KUKA KRL program: MyProgram_072().src

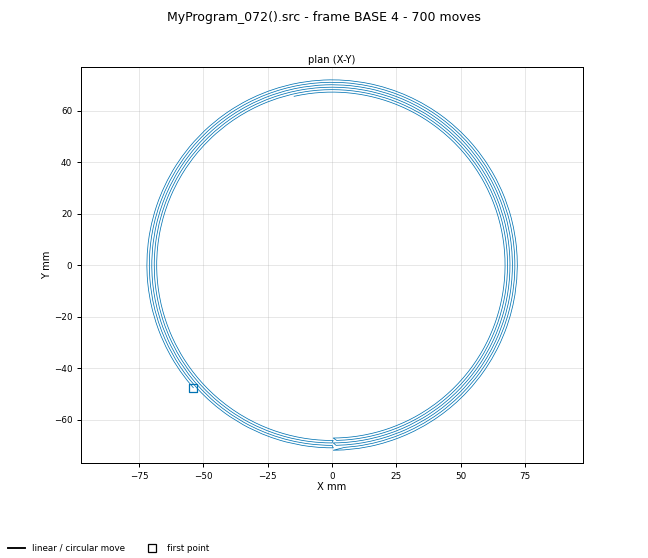
[picture p0: tool path of MyProgram_072().src in frame BASE 4, 700 of 700 moves have a stored position in this frame; points joined in program order, loops and branches not executed]
&ACCESS RVP
&REL 1
&PARAM TEMPLATE = C:\KRC\Roboter\Template\vorgabe
&PARAM EDITMASK = *
DEF MyProgram_072()
; ---- Setting reference (Base) ----
$BASE = BASE_DATA[4]

; --------------------------
; ---- Setting tool (TCP) ----
$TOOL = TOOL_DATA[3]
; --------------------------

$VEL.CP = VEL_APROX_PRINT
Startdeposition()
$VEL.CP = VEL_PRINT
LIN {X -53.9187,Y -47.6448,Z 77,A -144.3858,B 24.9058,C -2.2406,E1 24.8791,E2 228.8323} C_DIS
LIN {X -56.3583,Y -44.7314,Z 77,A -147.3901,B 24.9052,C -2.2481,E1 24.8738,E2 231.8326} C_DIS
LIN {X -58.9151,Y -41.3065,Z 77,A -151.2625,B 24.9054,C -2.2457,E1 24.8674,E2 235.7295} C_DIS
LIN {X -61.4241,Y -37.4729,Z 77,A -154.4026,B 24.9036,C -2.2665,E1 24.8627,E2 238.8358} C_DIS
LIN {X -62.7238,Y -35.2532,Z 77,A -157.5518,B 24.9052,C -2.2474,E1 24.8584,E2 242.0471} C_DIS
LIN {X -64.5699,Y -31.7477,Z 77,A -159.6161,B 24.9025,C -2.2803,E1 24.8558,E2 244.0442} C_DIS
LIN {X -66.4605,Y -27.5735,Z 77,A -163.4241,B 24.9019,C -2.2869,E1 24.8515,E2 247.8572} C_DIS
LIN {X -67.4022,Y -25.1814,Z 77,A -165.8052,B 24.902,C -2.2855,E1 24.8491,E2 250.2552} C_DIS
LIN {X -68.4094,Y -22.3006,Z 77,A -169.291,B 24.9034,C -2.2696,E1 24.8461,E2 253.7987} C_DIS
LIN {X -69.7872,Y -17.5225,Z 77,A -172.3901,B 24.9007,C -2.3002,E1 24.844,E2 256.8429} C_DIS
LIN {X -70.5609,Y -14.087,Z 77,A -174.6218,B 24.8989,C -2.3213,E1 24.8427,E2 259.0373} C_DIS
LIN {X -71.303,Y -9.6528,Z 77,A -178.4757,B 24.8985,C -2.3264,E1 24.841,E2 262.9021} C_DIS
LIN {X -71.6429,Y -6.6659,Z 77,A 179.1463,B 24.8978,C -2.3342,E1 24.8403,E2 265.2756} C_DIS
LIN {X -71.8296,Y -4.1964,Z 77,A 176.9907,B 24.8976,C -2.3365,E1 24.8399,E2 267.4388} C_DIS
LIN {X -71.951,Y -0.3995,Z 77,A 174.0055,B 24.8967,C -2.3469,E1 24.8398,E2 270.417} C_DIS
LIN {X -71.8201,Y 4.377,Z 77,A 169.8234,B 24.8963,C -2.3508,E1 24.8403,E2 274.615} C_DIS
LIN {X -71.4314,Y 8.6465,Z 77,A 166.8704,B 24.8945,C -2.3716,E1 24.8412,E2 277.5359} C_DIS
LIN {X -71.0021,Y 11.6566,Z 77,A 164.4409,B 24.8938,C -2.3791,E1 24.8422,E2 279.962} C_DIS
LIN {X -70.158,Y 15.9702,Z 77,A 161.2467,B 24.8922,C -2.3968,E1 24.8439,E2 283.1327} C_DIS
LIN {X -68.9886,Y 20.438,Z 77,A 157.304,B 24.8917,C -2.4024,E1 24.8468,E2 287.0849} C_DIS
LIN {X -68.1942,Y 22.9497,Z 77,A 155.1243,B 24.8913,C -2.4071,E1 24.8487,E2 289.266} C_DIS
LIN {X -67.3704,Y 25.267,Z 77,A 152.6721,B 24.8917,C -2.4023,E1 24.8511,E2 291.7435} C_DIS
LIN {X -65.9392,Y 28.7951,Z 77,A 148.9517,B 24.8922,C -2.3965,E1 24.8553,E2 295.4983} C_DIS
LIN {X -64.0236,Y 32.8348,Z 77,A 146.9975,B 24.8881,C -2.442,E1 24.8576,E2 297.3545} C_DIS
LIN {X -61.8148,Y 36.8256,Z 77,A 142.8596,B 24.8881,C -2.4411,E1 24.8633,E2 301.5161} C_DIS
LIN {X -60.5259,Y 38.9069,Z 77,A 140.6625,B 24.8881,C -2.4411,E1 24.8666,E2 303.7244} C_DIS
LIN {X -58.295,Y 42.1781,Z 77,A 137.1152,B 24.8881,C -2.4409,E1 24.8723,E2 307.2896} C_DIS
LIN {X -55.5018,Y 45.7902,Z 77,A 134.103,B 24.886,C -2.4642,E1 24.8775,E2 310.2602} C_DIS
LIN {X -53.6001,Y 48.0016,Z 77,A 131.2102,B 24.8867,C -2.4573,E1 24.8829,E2 313.1825} C_DIS
LIN {X -49.6348,Y 52.0931,Z 77,A 127.3776,B 24.8842,C -2.4839,E1 24.8903,E2 316.9677} C_DIS
LIN {X -47.6713,Y 53.8958,Z 77,A 124.8505,B 24.8846,C -2.4796,E1 24.8956,E2 319.5154} C_DIS
LIN {X -43.8735,Y 57.0285,Z 77,A 120.3096,B 24.8851,C -2.4739,E1 24.9056,E2 324.0866} C_DIS
LIN {X -41.0352,Y 59.1037,Z 77,A 118.2193,B 24.8831,C -2.4956,E1 24.9103,E2 326.1323} C_DIS
LIN {X -38.3583,Y 60.8757,Z 77,A 115.8538,B 24.8822,C -2.5048,E1 24.9158,E2 328.4836} C_DIS
LIN {X -34.6979,Y 63.0348,Z 77,A 112.3188,B 24.882,C -2.5073,E1 24.9244,E2 332.0233} C_DIS
LIN {X -32.2967,Y 64.2967,Z 77,A 110.0047,B 24.882,C -2.5072,E1 24.9301,E2 334.3439} C_DIS
LIN {X -29.0979,Y 65.8072,Z 77,A 106.6833,B 24.8827,C -2.4996,E1 24.9386,E2 337.6914} C_DIS
LIN {X -24.7486,Y 67.5622,Z 77,A 103.033,B 24.8821,C -2.5065,E1 24.9481,E2 341.3329} C_DIS
LIN {X -20.7016,Y 68.9104,Z 77,A 99.6928,B 24.8816,C -2.5117,E1 24.957,E2 344.6667} C_DIS
LIN {X -15.683,Y 70.2223,Z 77,A 95.9494,B 24.8803,C -2.5248,E1 24.9671,E2 348.384} C_DIS
LIN {X -12.4973,Y 70.8591,Z 77,A 93.0822,B 24.8808,C -2.5201,E1 24.975,E2 351.2656} C_DIS
LIN {X -7.8682,Y 71.5218,Z 77,A 89.6803,B 24.8798,C -2.5301,E1 24.9844,E2 354.6461} C_DIS
LIN {X -3.2799,Y 71.8778,Z 77,A 86.0502,B 24.8796,C -2.5325,E1 24.9945,E2 358.2719} C_DIS
LIN {X -0.9009,Y 71.9479,Z 77,A 83.3153,B 24.8815,C -2.5123,E1 25.0023,E2 361.0549} C_DIS
LIN {X 2.7139,Y 71.9018,Z 77,A 81.3961,B 24.8792,C -2.5363,E1 25.0075,E2 362.9166} C_DIS
LIN {X 6.8293,Y 71.6278,Z 77,A 77.9201,B 24.8797,C -2.5313,E1 25.0172,E2 366.4027} C_DIS
LIN {X 12.1948,Y 70.9121,Z 77,A 73.7586,B 24.8795,C -2.534,E1 25.0286,E2 370.5543} C_DIS
LIN {X 15.6992,Y 70.2197,Z 77,A 70.7865,B 24.8799,C -2.5294,E1 25.0368,E2 373.5334} C_DIS
LIN {X 19.6301,Y 69.2227,Z 77,A 67.0407,B 24.8813,C -2.5142,E1 25.0469,E2 377.3093} C_DIS
LIN {X 23.9385,Y 67.8535,Z 77,A 63.9687,B 24.8803,C -2.5248,E1 25.055,E2 380.3501} C_DIS
LIN {X 27.7756,Y 66.3753,Z 77,A 59.8788,B 24.8826,C -2.5004,E1 25.0657,E2 384.4886} C_DIS
LIN {X 31.1771,Y 64.8469,Z 77,A 57.9313,B 24.8805,C -2.5236,E1 25.0705,E2 386.3762} C_DIS
LIN {X 34.6789,Y 63.0444,Z 77,A 54.1919,B 24.8823,C -2.5036,E1 25.0798,E2 390.1524} C_DIS
LIN {X 38.4793,Y 60.8002,Z 77,A 51.0432,B 24.8819,C -2.5081,E1 25.0872,E2 393.2807} C_DIS
LIN {X 41.7065,Y 58.632,Z 77,A 48.2934,B 24.8815,C -2.5123,E1 25.0935,E2 396.011} C_DIS
LIN {X 43.7846,Y 57.097,Z 77,A 46.1388,B 24.8821,C -2.5061,E1 25.0984,E2 398.1726} C_DIS
LIN {X 46.6873,Y 54.7488,Z 77,A 42.9748,B 24.8831,C -2.4954,E1 25.1052,E2 401.3498} C_DIS
LIN {X 50.2229,Y 51.5263,Z 77,A 39.1466,B 24.8839,C -2.4872,E1 25.113,E2 405.1818} C_DIS
LIN {X 52.9217,Y 48.7488,Z 77,A 36.3509,B 24.8838,C -2.4884,E1 25.1184,E2 407.9624} C_DIS
LIN {X 54.7222,Y 46.7185,Z 77,A 34.2514,B 24.8841,C -2.4853,E1 25.1223,E2 410.06} C_DIS
LIN {X 56.9046,Y 44.0342,Z 77,A 31.1783,B 24.8855,C -2.47,E1 25.1277,E2 413.1549} C_DIS
LIN {X 59.7877,Y 40.0337,Z 77,A 27.4574,B 24.8859,C -2.466,E1 25.1336,E2 416.8672} C_DIS
LIN {X 62.2247,Y 36.1293,Z 77,A 23.0825,B 24.8886,C -2.4367,E1 25.14,E2 421.2888} C_DIS
LIN {X 63.774,Y 33.3177,Z 77,A 20.7832,B 24.8886,C -2.4369,E1 25.143,E2 423.5756} C_DIS
LIN {X 65.8578,Y 28.9817,Z 77,A 17.4795,B 24.8882,C -2.441,E1 25.1468,E2 426.8518} C_DIS
LIN {X 67.0447,Y 26.1186,Z 77,A 14.8515,B 24.8892,C -2.4294,E1 25.1496,E2 429.4926} C_DIS
LIN {X 68.871,Y 20.8324,Z 77,A 10.385,B 24.8905,C -2.4159,E1 25.1535,E2 433.9658} C_DIS
LIN {X 69.6052,Y 18.2306,Z 77,A 8.074,B 24.8915,C -2.405,E1 25.1552,E2 436.2893} C_DIS
LIN {X 70.4525,Y 14.6153,Z 77,A 5.2404,B 24.892,C -2.3994,E1 25.1569,E2 439.1195} C_DIS
LIN {X 71.252,Y 10.0146,Z 77,A 2.1561,B 24.8914,C -2.406,E1 25.1583,E2 442.1703} C_DIS
LIN {X 71.6054,Y 7.0466,Z 77,A -0.7092,B 24.8933,C -2.3847,E1 25.1592,E2 445.0689} C_DIS
LIN {X 71.868,Y 3.4604,Z 77,A -3.831,B 24.8948,C -2.3683,E1 25.1597,E2 448.2109} C_DIS
LIN {X 71.9513,Y -0.3429,Z 77,A -6.9056,B 24.8957,C -2.3574,E1 25.1597,E2 451.293} C_DIS
LIN {X 71.7394,Y -5.5341,Z 77,A -11.1078,B 24.897,C -2.3424,E1 25.159,E2 455.5057} C_DIS
LIN {X 71.0278,Y -11.5028,Z 77,A -16.3322,B 24.8995,C -2.3149,E1 25.1569,E2 460.7642} C_DIS
LIN {X 70.2523,Y -15.5498,Z 77,A -18.4428,B 24.8975,C -2.3377,E1 25.1558,E2 462.8086} C_DIS
LIN {X 69.2248,Y -19.6231,Z 77,A -21.5617,B 24.8978,C -2.3337,E1 25.1536,E2 465.919} C_DIS
LIN {X 67.943,Y -23.6835,Z 77,A -24.9418,B 24.8987,C -2.3235,E1 25.1508,E2 469.304} C_DIS
LIN {X 67.0842,Y -26.0181,Z 77,A -27.7452,B 24.9013,C -2.2941,E1 25.1479,E2 472.1614} C_DIS
LIN {X 65.4629,Y -29.864,Z 77,A -30.3132,B 24.9003,C -2.3055,E1 25.1451,E2 474.6883} C_DIS
LIN {X 64.2104,Y -32.4692,Z 77,A -33.0533,B 24.9019,C -2.2863,E1 25.1417,E2 477.4591} C_DIS
LIN {X 61.9999,Y -36.5125,Z 77,A -36.9921,B 24.9035,C -2.2682,E1 25.1362,E2 481.4202} C_DIS
LIN {X 59.5766,Y -40.3456,Z 77,A -40.253,B 24.9035,C -2.268,E1 25.1312,E2 484.6654} C_DIS
LIN {X 57.5966,Y -43.1251,Z 77,A -42.6994,B 24.9035,C -2.2683,E1 25.1272,E2 487.0993} C_DIS
LIN {X 54.3876,Y -47.1084,Z 77,A -46.7073,B 24.9042,C -2.2595,E1 25.1201,E2 491.1094} C_DIS
LIN {X 51.4117,Y -50.3396,Z 77,A -50.3462,B 24.9053,C -2.2469,E1 25.1132,E2 494.7622} C_DIS
LIN {X 48.408,Y -53.2321,Z 77,A -53.6707,B 24.906,C -2.2391,E1 25.1064,E2 498.0915} C_DIS
LIN {X 45.7832,Y -55.5077,Z 77,A -56.6724,B 24.907,C -2.2264,E1 25.0999,E2 501.1116} C_DIS
LIN {X 43.0423,Y -57.6588,Z 77,A -59.2217,B 24.907,C -2.2268,E1 25.0943,E2 503.6508} C_DIS
LIN {X 39.929,Y -59.8578,Z 77,A -62.2452,B 24.9075,C -2.221,E1 25.0873,E2 506.6776} C_DIS
LIN {X 35.9325,Y -62.3378,Z 77,A -66.2637,B 24.9087,C -2.2068,E1 25.0777,E2 510.7173} C_DIS
LIN {X 31.9087,Y -64.4901,Z 77,A -69.8151,B 24.909,C -2.203,E1 25.0689,E2 514.2679} C_DIS
LIN {X 28.8413,Y -65.919,Z 77,A -72.2737,B 24.9088,C -2.2052,E1 25.0626,E2 516.7151} C_DIS
LIN {X 26.0215,Y -67.0829,Z 77,A -74.4572,B 24.9085,C -2.2084,E1 25.057,E2 518.8861} C_DIS
LIN {X 23.2742,Y -68.0848,Z 77,A -77.7414,B 24.9108,C -2.1802,E1 25.0482,E2 522.2308} C_DIS
LIN {X 19.8136,Y -69.1708,Z 77,A -79.4127,B 24.9085,C -2.2091,E1 25.0439,E2 523.8305} C_DIS
LIN {X 16.8729,Y -69.9462,Z 77,A -82.0355,B 24.9091,C -2.2013,E1 25.0368,E2 526.4678} C_DIS
LIN {X 14.9547,Y -70.3821,Z 77,A -83.9899,B 24.9101,C -2.1896,E1 25.0314,E2 528.4473} C_DIS
LIN {X 10.5522,Y -71.1757,Z 77,A -87.9511,B 24.9111,C -2.1767,E1 25.0204,E2 532.4353} C_DIS
LIN {X 4.5761,Y -71.8072,Z 77,A -92.5167,B 24.9109,C -2.1799,E1 25.0077,E2 536.9906} C_DIS
LIN {X 0.4767,Y -71.9366,Z 77,A -94.7077,B 24.9086,C -2.2068,E1 25.0018,E2 539.1173} C_DIS
Enddeposition()
LIN {X 0.4767,Y -71.9366,Z 77,A -94.7077,B 24.9086,C -2.2068,E1 25.0018,E2 539.1173} C_DIS
Startdeposition()
$VEL.CP = VEL_PRINT
LIN {X 4.8028,Y -70.8374,Z 77,A -90.3844,B 24.9054,C -2.2459,E1 25.0141,E2 534.7027} C_DIS
LIN {X 9.797,Y -70.3212,Z 77,A -87.1467,B 24.907,C -2.227,E1 25.0229,E2 531.5122} C_DIS
LIN {X 11.8985,Y -69.9962,Z 77,A -84.5588,B 24.9049,C -2.2512,E1 25.0302,E2 528.8694} C_DIS
LIN {X 15.8769,Y -69.2021,Z 77,A -81.1578,B 24.9044,C -2.2576,E1 25.0395,E2 525.4579} C_DIS
LIN {X 19.7248,Y -68.2062,Z 77,A -78.0106,B 24.9042,C -2.2594,E1 25.048,E2 522.3116} C_DIS
LIN {X 24.4836,Y -66.6453,Z 77,A -74.1651,B 24.9042,C -2.2592,E1 25.0581,E2 518.4743} C_DIS
LIN {X 28.2316,Y -65.1461,Z 77,A -70.4132,B 24.9027,C -2.2774,E1 25.0678,E2 514.6881} C_DIS
LIN {X 31.7235,Y -63.5191,Z 77,A -68.2259,B 24.9044,C -2.2572,E1 25.0732,E2 512.5547} C_DIS
LIN {X 35.7437,Y -61.348,Z 77,A -64.1814,B 24.903,C -2.2734,E1 25.0831,E2 508.4836} C_DIS
LIN {X 39.7187,Y -58.8511,Z 77,A -61.0974,B 24.9041,C -2.2613,E1 25.0902,E2 505.4384} C_DIS
LIN {X 42.4392,Y -56.9209,Z 77,A -58.4529,B 24.9037,C -2.2654,E1 25.0962,E2 502.7933} C_DIS
LIN {X 44.0637,Y -55.6723,Z 77,A -55.8093,B 24.9011,C -2.2965,E1 25.1022,E2 500.086} C_DIS
LIN {X 47.6747,Y -52.6136,Z 77,A -52.5448,B 24.9016,C -2.2896,E1 25.109,E2 496.8507} C_DIS
LIN {X 50.1301,Y -50.2801,Z 77,A -49.8672,B 24.9012,C -2.2945,E1 25.1143,E2 494.1727} C_DIS
LIN {X 52.5803,Y -47.7124,Z 77,A -46.9276,B 24.9004,C -2.3037,E1 25.1199,E2 491.2242} C_DIS
LIN {X 55.7281,Y -43.9931,Z 77,A -43.3118,B 24.9004,C -2.305,E1 25.1263,E2 487.6221} C_DIS
LIN {X 57.3663,Y -41.8346,Z 77,A -40.9757,B 24.8994,C -2.3151,E1 25.1302,E2 485.2733} C_DIS
LIN {X 59.8557,Y -38.1883,Z 77,A -37.1704,B 24.898,C -2.3318,E1 25.1362,E2 481.4474} C_DIS
LIN {X 62.6104,Y -33.4832,Z 77,A -33.0702,B 24.8976,C -2.3359,E1 25.1418,E2 477.3589} C_DIS
LIN {X 64.9521,Y -28.6765,Z 77,A -28.9167,B 24.8969,C -2.344,E1 25.1468,E2 473.2084} C_DIS
LIN {X 66.7625,Y -24.1621,Z 77,A -24.9117,B 24.8957,C -2.3582,E1 25.1509,E2 469.1921} C_DIS
LIN {X 68.1104,Y -20.0502,Z 77,A -21.6688,B 24.8953,C -2.3619,E1 25.1536,E2 465.9591} C_DIS
LIN {X 68.9713,Y -16.8514,Z 77,A -18.6869,B 24.8938,C -2.3791,E1 25.1557,E2 462.9537} C_DIS
LIN {X 69.826,Y -12.8621,Z 77,A -15.6337,B 24.8935,C -2.3826,E1 25.1574,E2 459.91} C_DIS
LIN {X 70.2378,Y -10.3839,Z 77,A -12.2641,B 24.8894,C -2.4278,E1 25.1588,E2 456.4534} C_DIS
LIN {X 70.7674,Y -5.7434,Z 77,A -10.2321,B 24.8928,C -2.3897,E1 25.1593,E2 454.5236} C_DIS
LIN {X 70.9871,Y -1.3604,Z 77,A -6.2727,B 24.8907,C -2.4128,E1 25.1598,E2 450.5329} C_DIS
LIN {X 70.983,Y 1.5815,Z 77,A -3.6125,B 24.8893,C -2.4286,E1 25.1597,E2 447.8514} C_DIS
LIN {X 70.8141,Y 5.1488,Z 77,A -0.9641,B 24.8891,C -2.431,E1 25.1592,E2 445.2131} C_DIS
LIN {X 70.4749,Y 8.6274,Z 77,A 1.5523,B 24.8891,C -2.4311,E1 25.1585,E2 442.7112} C_DIS
LIN {X 70.1756,Y 10.789,Z 77,A 3.8082,B 24.8873,C -2.4507,E1 25.1575,E2 440.4222} C_DIS
LIN {X 69.5035,Y 14.5026,Z 77,A 6.5362,B 24.8873,C -2.451,E1 25.1561,E2 437.7094} C_DIS
LIN {X 68.834,Y 17.4059,Z 77,A 8.6114,B 24.8874,C -2.449,E1 25.1548,E2 435.6511} C_DIS
LIN {X 68.2901,Y 19.4287,Z 77,A 11.0027,B 24.8851,C -2.474,E1 25.1529,E2 433.2144} C_DIS
LIN {X 66.7102,Y 24.3056,Z 77,A 14.6305,B 24.8853,C -2.4716,E1 25.1497,E2 429.6126} C_DIS
LIN {X 64.9023,Y 28.7903,Z 77,A 18.5475,B 24.8843,C -2.4832,E1 25.1455,E2 425.69} C_DIS
LIN {X 63.9127,Y 30.9228,Z 77,A 20.6659,B 24.8832,C -2.4947,E1 25.1429,E2 423.5558} C_DIS
LIN {X 62.7651,Y 33.1899,Z 77,A 22.6008,B 24.883,C -2.497,E1 25.1405,E2 421.6256} C_DIS
LIN {X 59.7783,Y 38.3089,Z 77,A 27.1898,B 24.8823,C -2.504,E1 25.1339,E2 417.0434} C_DIS
LIN {X 57.097,Y 42.2025,Z 77,A 30.7011,B 24.8823,C -2.5051,E1 25.1283,E2 413.5469} C_DIS
LIN {X 54.6084,Y 45.3755,Z 77,A 33.7833,B 24.8819,C -2.508,E1 25.123,E2 410.4722} C_DIS
LIN {X 52.0939,Y 48.2426,Z 77,A 37.6886,B 24.8791,C -2.5376,E1 25.1156,E2 406.5143} C_DIS
LIN {X 49.5448,Y 50.8573,Z 77,A 41.0558,B 24.8774,C -2.5553,E1 25.1089,E2 403.1193} C_DIS
LIN {X 47.0744,Y 53.1521,Z 77,A 42.7817,B 24.8795,C -2.5335,E1 25.1054,E2 401.4521} C_DIS
LIN {X 43.9657,Y 55.7497,Z 77,A 45.6849,B 24.8799,C -2.5297,E1 25.0993,E2 398.5689} C_DIS
LIN {X 40.834,Y 58.0839,Z 77,A 49.1667,B 24.8785,C -2.544,E1 25.0914,E2 395.0659} C_DIS
LIN {X 38.929,Y 59.3765,Z 77,A 51.056,B 24.8781,C -2.5478,E1 25.087,E2 393.1738} C_DIS
LIN {X 36.7766,Y 60.7331,Z 77,A 53.5141,B 24.8768,C -2.5617,E1 25.0811,E2 390.6906} C_DIS
LIN {X 33.4485,Y 62.6267,Z 77,A 56.6188,B 24.8764,C -2.5663,E1 25.0735,E2 387.584} C_DIS
LIN {X 30.2857,Y 64.2177,Z 77,A 59.5792,B 24.8758,C -2.5724,E1 25.066,E2 384.6169} C_DIS
LIN {X 27.2313,Y 65.5714,Z 77,A 62.7226,B 24.8743,C -2.587,E1 25.0579,E2 381.446} C_DIS
LIN {X 23.9804,Y 66.8288,Z 77,A 64.7854,B 24.876,C -2.5699,E1 25.0526,E2 379.4283} C_DIS
LIN {X 20.5721,Y 67.954,Z 77,A 68.4447,B 24.8739,C -2.592,E1 25.0427,E2 375.7231} C_DIS
LIN {X 17.1154,Y 68.9069,Z 77,A 70.2141,B 24.8765,C -2.5646,E1 25.0381,E2 374.0214} C_DIS
LIN {X 15.0478,Y 69.3872,Z 77,A 72.237,B 24.8757,C -2.5734,E1 25.0325,E2 371.9804} C_DIS
LIN {X 11.7294,Y 70.0245,Z 77,A 75.5579,B 24.8741,C -2.5896,E1 25.0233,E2 368.6246} C_DIS
LIN {X 7.2897,Y 70.6249,Z 77,A 78.5804,B 24.8755,C -2.5752,E1 25.015,E2 365.6386} C_DIS
LIN {X 4.0751,Y 70.8832,Z 77,A 81.3131,B 24.8752,C -2.5785,E1 25.0074,E2 362.8992} C_DIS
LIN {X -0.8301,Y 70.9963,Z 77,A 85.2568,B 24.8752,C -2.5774,E1 24.9964,E2 358.9585} C_DIS
LIN {X -4.2337,Y 70.8744,Z 77,A 87.9354,B 24.8755,C -2.5748,E1 24.9889,E2 356.2855} C_DIS
LIN {X -8.0718,Y 70.54,Z 77,A 91.9066,B 24.8736,C -2.5945,E1 24.9778,E2 352.2651} C_DIS
LIN {X -11.8134,Y 70.0105,Z 77,A 93.8627,B 24.8764,C -2.5655,E1 24.9726,E2 350.3761} C_DIS
LIN {X -14.2047,Y 69.5647,Z 77,A 96.5684,B 24.8748,C -2.582,E1 24.965,E2 347.6282} C_DIS
LIN {X -17.5794,Y 68.7894,Z 77,A 99.5675,B 24.8746,C -2.5843,E1 24.9569,E2 344.6193} C_DIS
LIN {X -20.826,Y 67.8773,Z 77,A 101.2258,B 24.8774,C -2.5557,E1 24.9526,E2 343.0262} C_DIS
LIN {X -23.8652,Y 66.87,Z 77,A 104.5093,B 24.8761,C -2.5693,E1 24.9439,E2 339.7042} C_DIS
LIN {X -27.2429,Y 65.5661,Z 77,A 107.7082,B 24.8758,C -2.5719,E1 24.9356,E2 336.492} C_DIS
LIN {X -31.3437,Y 63.7074,Z 77,A 111.4378,B 24.8761,C -2.5685,E1 24.9262,E2 332.7608} C_DIS
LIN {X -34.2876,Y 62.1732,Z 77,A 113.157,B 24.8787,C -2.5415,E1 24.9221,E2 331.1012} C_DIS
LIN {X -37.7438,Y 60.1369,Z 77,A 116.3124,B 24.8795,C -2.5338,E1 24.9146,E2 327.9546} C_DIS
LIN {X -39.5422,Y 58.9706,Z 77,A 118.8783,B 24.8779,C -2.5498,E1 24.9085,E2 325.3419} C_DIS
LIN {X -43.189,Y 56.3538,Z 77,A 122.1065,B 24.8795,C -2.5333,E1 24.9013,E2 322.1416} C_DIS
LIN {X -45.8828,Y 54.1833,Z 77,A 124.8725,B 24.8802,C -2.5266,E1 24.8953,E2 319.381} C_DIS
LIN {X -48.2766,Y 52.0627,Z 77,A 127.8202,B 24.8799,C -2.5291,E1 24.8892,E2 316.4155} C_DIS
LIN {X -51.0045,Y 49.3921,Z 77,A 130.6169,B 24.8812,C -2.5153,E1 24.8838,E2 313.6398} C_DIS
LIN {X -53.4104,Y 46.7798,Z 77,A 133.3965,B 24.8821,C -2.5063,E1 24.8786,E2 310.8696} C_DIS
LIN {X -55.4307,Y 44.3693,Z 77,A 136.8622,B 24.8807,C -2.5207,E1 24.8724,E2 307.3533} C_DIS
LIN {X -57.6702,Y 41.415,Z 77,A 138.8839,B 24.8836,C -2.4908,E1 24.8692,E2 305.3931} C_DIS
LIN {X -60.4569,Y 37.231,Z 77,A 142.8404,B 24.8848,C -2.4773,E1 24.8632,E2 301.4489} C_DIS
LIN {X -63.052,Y 32.6434,Z 77,A 147.2087,B 24.8857,C -2.4676,E1 24.8572,E2 297.0808} C_DIS
LIN {X -64.9825,Y 28.6067,Z 77,A 150.6329,B 24.8871,C -2.4529,E1 24.8532,E2 293.6732} C_DIS
LIN {X -66.6443,Y 24.4861,Z 77,A 154.5456,B 24.8874,C -2.4492,E1 24.8491,E2 289.7474} C_DIS
LIN {X -67.5853,Y 21.7542,Z 77,A 156.9132,B 24.888,C -2.4428,E1 24.847,E2 287.3815} C_DIS
LIN {X -68.7027,Y 17.9166,Z 77,A 160.6729,B 24.8878,C -2.4446,E1 24.8442,E2 283.5957} C_DIS
LIN {X -69.5361,Y 14.3437,Z 77,A 162.9939,B 24.89,C -2.4212,E1 24.8429,E2 281.317} C_DIS
LIN {X -70.0772,Y 11.4141,Z 77,A 165.8284,B 24.8898,C -2.4231,E1 24.8415,E2 278.4613} C_DIS
LIN {X -70.4964,Y 8.444,Z 77,A 167.9157,B 24.8912,C -2.4081,E1 24.8408,E2 276.3973} C_DIS
LIN {X -70.7959,Y 5.3874,Z 77,A 170.5761,B 24.8915,C -2.4042,E1 24.8401,E2 273.7302} C_DIS
LIN {X -70.9416,Y 2.875,Z 77,A 172.7534,B 24.8918,C -2.401,E1 24.8398,E2 271.5474} C_DIS
LIN {X -70.9975,Y -0.6252,Z 77,A 175.6411,B 24.8925,C -2.3934,E1 24.8398,E2 268.6604} C_DIS
LIN {X -70.813,Y -5.1646,Z 77,A 179.2227,B 24.8937,C -2.3799,E1 24.8404,E2 265.0894} C_DIS
LIN {X -70.5239,Y -8.2094,Z 77,A -178.3146,B 24.8944,C -2.3721,E1 24.8411,E2 262.6306} C_DIS
LIN {X -69.6888,Y -13.5831,Z 77,A -173.8956,B 24.8956,C -2.3592,E1 24.8431,E2 258.2163} C_DIS
LIN {X -68.8541,Y -17.3279,Z 77,A -169.5554,B 24.8939,C -2.3778,E1 24.8461,E2 253.8063} C_DIS
LIN {X -67.5209,Y -21.9535,Z 77,A -167.1097,B 24.8978,C -2.3339,E1 24.8481,E2 251.4515} C_DIS
LIN {X -66.2069,Y -25.6436,Z 77,A -163.5717,B 24.8978,C -2.3331,E1 24.8515,E2 247.8953} C_DIS
LIN {X -65.009,Y -28.546,Z 77,A -161.0325,B 24.8985,C -2.3261,E1 24.8543,E2 245.3589} C_DIS
LIN {X -63.533,Y -31.6954,Z 77,A -157.8695,B 24.8985,C -2.3264,E1 24.8582,E2 242.178} C_DIS
LIN {X -60.8132,Y -36.6447,Z 77,A -154.1487,B 24.9012,C -2.2953,E1 24.8632,E2 238.5118} C_DIS
LIN {X -59.1818,Y -39.2243,Z 77,A -151.0211,B 24.9004,C -2.3042,E1 24.868,E2 235.3474} C_DIS
LIN {X -57.279,Y -41.9539,Z 77,A -148.7375,B 24.9018,C -2.2884,E1 24.8717,E2 233.0903} C_DIS
LIN {X -55.4855,Y -44.3001,Z 77,A -145.9511,B 24.9014,C -2.292,E1 24.8765,E2 230.2821} C_DIS
LIN {X -52.2898,Y -48.0291,Z 77,A -142.593,B 24.9034,C -2.2692,E1 24.8826,E2 226.9633} C_DIS
LIN {X -50.6569,Y -49.7487,Z 77,A -139.9543,B 24.9023,C -2.282,E1 24.8878,E2 224.2829} C_DIS
LIN {X -48.1592,Y -52.1701,Z 77,A -137.0442,B 24.9026,C -2.2787,E1 24.8938,E2 221.3685} C_DIS
LIN {X -45.0911,Y -54.8447,Z 77,A -133.8399,B 24.9033,C -2.2707,E1 24.9006,E2 218.1711} C_DIS
LIN {X -41.6123,Y -57.5285,Z 77,A -130.8901,B 24.905,C -2.2504,E1 24.9071,E2 215.259} C_DIS
LIN {X -39.7167,Y -58.8524,Z 77,A -128.2557,B 24.9037,C -2.2658,E1 24.9133,E2 212.5792} C_DIS
LIN {X -34.5305,Y -62.0376,Z 77,A -124.1182,B 24.9059,C -2.2401,E1 24.9231,E2 208.4901} C_DIS
LIN {X -32.5849,Y -63.0819,Z 77,A -121.6017,B 24.9046,C -2.2556,E1 24.9294,E2 205.9298} C_DIS
LIN {X -27.2101,Y -65.5803,Z 77,A -117.5797,B 24.9066,C -2.2318,E1 24.9396,E2 201.9548} C_DIS
LIN {X -23.5533,Y -66.9793,Z 77,A -113.2832,B 24.9044,C -2.2571,E1 24.951,E2 197.5893} C_DIS
LIN {X -20.1562,Y -68.0789,Z 77,A -111.3901,B 24.9067,C -2.2305,E1 24.9559,E2 195.7564} C_DIS
LIN {X -17.8656,Y -68.7159,Z 77,A -108.6876,B 24.9051,C -2.2489,E1 24.9633,E2 193.0061} C_DIS
LIN {X -11.6709,Y -70.0343,Z 77,A -104.3681,B 24.907,C -2.2269,E1 24.975,E2 188.7339} C_DIS
LIN {X -9.1478,Y -70.4083,Z 77,A -101.7458,B 24.9058,C -2.2408,E1 24.9824,E2 186.0766} C_DIS
LIN {X -5.4062,Y -70.7944,Z 77,A -98.3265,B 24.905,C -2.2506,E1 24.992,E2 182.6326} C_DIS
LIN {X -2.0223,Y -70.9714,Z 77,A -96.5275,B 24.907,C -2.2268,E1 24.9968,E2 180.8898} C_DIS
LIN {X 0.4624,Y -70.9986,Z 77,A -95.4279,B 24.9089,C -2.2041,E1 24.9998,E2 179.8439} C_DIS
Enddeposition()
LIN {X 0.4624,Y -70.9986,Z 77,A -95.4279,B 24.9089,C -2.2041,E1 24.9998,E2 179.8439} C_DIS
Startdeposition()
$VEL.CP = VEL_PRINT
LIN {X 0.022,Y -70.049,Z 77,A -95.9251,B 24.9078,C -2.2173,E1 24.9984,E2 180.3097} C_DIS
LIN {X -2.3046,Y -70.0101,Z 77,A -98.1613,B 24.9085,C -2.2089,E1 24.9921,E2 182.5663} C_DIS
LIN {X -7.0392,Y -69.6937,Z 77,A -101.6888,B 24.9077,C -2.2177,E1 24.9824,E2 186.0744} C_DIS
LIN {X -10.1885,Y -69.3038,Z 77,A -104.2753,B 24.9077,C -2.2184,E1 24.9752,E2 188.6612} C_DIS
LIN {X -14.4831,Y -68.5354,Z 77,A -108.1851,B 24.9083,C -2.2115,E1 24.9644,E2 192.5917} C_DIS
LIN {X -18.326,Y -67.6082,Z 77,A -111.0923,B 24.9075,C -2.2212,E1 24.9566,E2 195.4801} C_DIS
LIN {X -22.3353,Y -66.3916,Z 77,A -114.8329,B 24.9079,C -2.2163,E1 24.9466,E2 199.239} C_DIS
LIN {X -25.9611,Y -65.0605,Z 77,A -117.6264,B 24.9069,C -2.2278,E1 24.9394,E2 202.011} C_DIS
LIN {X -29.1631,Y -63.6892,Z 77,A -120.6728,B 24.907,C -2.2263,E1 24.9316,E2 205.0684} C_DIS
LIN {X -32.2878,Y -62.164,Z 77,A -123.3936,B 24.9065,C -2.2326,E1 24.9248,E2 207.7814} C_DIS
LIN {X -34.3561,Y -61.0444,Z 77,A -125.7546,B 24.9071,C -2.2252,E1 24.919,E2 210.1671} C_DIS
LIN {X -39.0448,Y -58.1574,Z 77,A -129.4882,B 24.9051,C -2.2496,E1 24.9103,E2 213.8542} C_DIS
LIN {X -42.6178,Y -55.5919,Z 77,A -133.492,B 24.9053,C -2.2464,E1 24.9013,E2 217.8798} C_DIS
LIN {X -45.1547,Y -53.5527,Z 77,A -135.7828,B 24.9042,C -2.2597,E1 24.8963,E2 220.1475} C_DIS
LIN {X -47.0139,Y -51.927,Z 77,A -138.1635,B 24.9046,C -2.2555,E1 24.8913,E2 222.5477} C_DIS
LIN {X -50.6999,Y -48.336,Z 77,A -142.0716,B 24.9032,C -2.271,E1 24.8836,E2 226.4355} C_DIS
LIN {X -53.5232,Y -45.1892,Z 77,A -145.9887,B 24.9035,C -2.2685,E1 24.8764,E2 230.376} C_DIS
LIN {X -55.6876,Y -42.4935,Z 77,A -148.8959,B 24.903,C -2.2734,E1 24.8714,E2 233.2852} C_DIS
LIN {X -59.2312,Y -37.3962,Z 77,A -153.7672,B 24.9016,C -2.2906,E1 24.8638,E2 238.1396} C_DIS
LIN {X -60.3903,Y -35.4923,Z 77,A -155.9166,B 24.9018,C -2.2883,E1 24.8607,E2 240.3056} C_DIS
LIN {X -62.5754,Y -31.4833,Z 77,A -159.3659,B 24.9004,C -2.3046,E1 24.8562,E2 243.7345} C_DIS
LIN {X -63.6284,Y -29.2954,Z 77,A -161.6023,B 24.9004,C -2.3047,E1 24.8536,E2 245.9828} C_DIS
LIN {X -65.7401,Y -24.1864,Z 77,A -165.8865,B 24.8988,C -2.3228,E1 24.8491,E2 250.2478} C_DIS
LIN {X -66.5675,Y -21.8069,Z 77,A -168.3011,B 24.8989,C -2.3213,E1 24.847,E2 252.6797} C_DIS
LIN {X -67.9209,Y -17.1334,Z 77,A -171.8826,B 24.8971,C -2.3417,E1 24.8444,E2 256.2333} C_DIS
LIN {X -68.7338,Y -13.5069,Z 77,A -174.6839,B 24.8958,C -2.356,E1 24.8427,E2 259.0168} C_DIS
LIN {X -69.3006,Y -10.2108,Z 77,A -177.7743,B 24.8958,C -2.3569,E1 24.8413,E2 262.1235} C_DIS
LIN {X -69.6533,Y -7.4259,Z 77,A 179.8553,B 24.8953,C -2.3625,E1 24.8405,E2 264.4947} C_DIS
LIN {X -69.9218,Y -4.2145,Z 77,A 177.095,B 24.8948,C -2.3682,E1 24.84,E2 267.2581} C_DIS
LIN {X -70.044,Y -0.851,Z 77,A 174.4692,B 24.8937,C -2.3796,E1 24.8398,E2 269.8725} C_DIS
LIN {X -70.0249,Y 1.7981,Z 77,A 172.1227,B 24.8935,C -2.3827,E1 24.8399,E2 272.2257} C_DIS
LIN {X -69.7534,Y 6.4158,Z 77,A 168.6122,B 24.8919,C -2.4005,E1 24.8406,E2 275.7148} C_DIS
LIN {X -69.5001,Y 8.7465,Z 77,A 166.156,B 24.8923,C -2.3952,E1 24.8414,E2 278.1983} C_DIS
LIN {X -68.7113,Y 13.6225,Z 77,A 162.6055,B 24.8903,C -2.4182,E1 24.8431,E2 281.7148} C_DIS
LIN {X -67.9681,Y 16.9458,Z 77,A 159.2799,B 24.8905,C -2.4156,E1 24.8452,E2 285.0662} C_DIS
LIN {X -66.8083,Y 21.0583,Z 77,A 155.3482,B 24.8903,C -2.4173,E1 24.8485,E2 289.0164} C_DIS
LIN {X -65.6705,Y 24.3772,Z 77,A 152.9474,B 24.8886,C -2.4358,E1 24.8507,E2 291.3866} C_DIS
LIN {X -64.3712,Y 27.6264,Z 77,A 150.5991,B 24.8869,C -2.4553,E1 24.8532,E2 293.7014} C_DIS
LIN {X -62.9153,Y 30.7969,Z 77,A 147.3349,B 24.8869,C -2.455,E1 24.8571,E2 296.9841} C_DIS
LIN {X -60.4658,Y 35.3651,Z 77,A 143.2762,B 24.8854,C -2.471,E1 24.8625,E2 301.0258} C_DIS
LIN {X -58.6526,Y 38.2957,Z 77,A 140.0355,B 24.8855,C -2.4699,E1 24.8674,E2 304.2857} C_DIS
LIN {X -57.0452,Y 40.6515,Z 77,A 136.8467,B 24.8866,C -2.458,E1 24.8727,E2 307.5184} C_DIS
LIN {X -54.2908,Y 44.2635,Z 77,A 134.2615,B 24.8835,C -2.4918,E1 24.8771,E2 310.0352} C_DIS
LIN {X -51.6515,Y 47.3162,Z 77,A 130.8108,B 24.883,C -2.4968,E1 24.8835,E2 313.4894} C_DIS
LIN {X -49.0592,Y 49.9989,Z 77,A 127.4909,B 24.8829,C -2.4982,E1 24.89,E2 316.8199} C_DIS
LIN {X -46.4565,Y 52.4273,Z 77,A 125.1986,B 24.8809,C -2.5184,E1 24.8947,E2 319.0734} C_DIS
LIN {X -43.9711,Y 54.5267,Z 77,A 122.1973,B 24.8811,C -2.5167,E1 24.9012,E2 322.0901} C_DIS
LIN {X -40.7151,Y 56.999,Z 77,A 118.3178,B 24.8816,C -2.5117,E1 24.91,E2 325.9952} C_DIS
LIN {X -37.4944,Y 59.169,Z 77,A 115.5273,B 24.8802,C -2.5262,E1 24.9165,E2 328.7601} C_DIS
LIN {X -34.1736,Y 61.1463,Z 77,A 112.2559,B 24.8799,C -2.5293,E1 24.9244,E2 332.0338} C_DIS
LIN {X -30.7486,Y 62.9395,Z 77,A 109.5066,B 24.8785,C -2.5437,E1 24.9312,E2 334.7564} C_DIS
LIN {X -26.1366,Y 64.9897,Z 77,A 105.4728,B 24.8778,C -2.5518,E1 24.9415,E2 338.7804} C_DIS
LIN {X -22.9758,Y 66.173,Z 77,A 102.3594,B 24.8782,C -2.5472,E1 24.9497,E2 341.9109} C_DIS
LIN {X -18.3354,Y 67.6056,Z 77,A 98.5723,B 24.8774,C -2.5558,E1 24.9598,E2 345.6839} C_DIS
LIN {X -14.4248,Y 68.5471,Z 77,A 95.1811,B 24.8774,C -2.5564,E1 24.969,E2 349.0781} C_DIS
LIN {X -11.2016,Y 69.1473,Z 77,A 91.9461,B 24.8784,C -2.5454,E1 24.978,E2 352.3424} C_DIS
LIN {X -5.422,Y 69.8379,Z 77,A 87.7334,B 24.8769,C -2.5608,E1 24.9896,E2 356.5208} C_DIS
LIN {X -2.4339,Y 70.0061,Z 77,A 85.3415,B 24.8767,C -2.563,E1 24.9963,E2 358.9081} C_DIS
LIN {X -0.2691,Y 70.0475,Z 77,A 83.2783,B 24.8773,C -2.5564,E1 25.0021,E2 360.9871} C_DIS
LIN {X 4.4587,Y 69.9063,Z 77,A 79.6612,B 24.8767,C -2.5627,E1 25.0121,E2 364.5881} C_DIS
LIN {X 7.3719,Y 69.6589,Z 77,A 77.2788,B 24.8767,C -2.5627,E1 25.0187,E2 366.9691} C_DIS
LIN {X 11.2639,Y 69.1369,Z 77,A 73.779,B 24.8775,C -2.5547,E1 25.0284,E2 370.4846} C_DIS
LIN {X 14.6984,Y 68.4888,Z 77,A 71.2718,B 24.8768,C -2.5622,E1 25.0352,E2 372.971} C_DIS
LIN {X 16.9181,Y 67.9749,Z 77,A 68.9804,B 24.8779,C -2.5505,E1 25.0415,E2 375.2868} C_DIS
LIN {X 21.5367,Y 66.6549,Z 77,A 65.3997,B 24.8773,C -2.5564,E1 25.051,E2 378.8472} C_DIS
LIN {X 24.8831,Y 65.4793,Z 77,A 62.4686,B 24.8776,C -2.553,E1 25.0587,E2 381.7803} C_DIS
LIN {X 27.3602,Y 64.4837,Z 77,A 60.3467,B 24.8777,C -2.5523,E1 25.0642,E2 383.8989} C_DIS
LIN {X 30.1415,Y 63.2316,Z 77,A 57.8996,B 24.8779,C -2.5506,E1 25.0704,E2 386.3438} C_DIS
LIN {X 33.2243,Y 61.6675,Z 77,A 54.8857,B 24.8787,C -2.5422,E1 25.0779,E2 389.3692} C_DIS
LIN {X 36.5599,Y 59.7504,Z 77,A 51.9873,B 24.8785,C -2.5441,E1 25.0848,E2 392.2542} C_DIS
LIN {X 38.462,Y 58.5439,Z 77,A 49.9572,B 24.8792,C -2.5364,E1 25.0896,E2 394.296} C_DIS
LIN {X 41.1868,Y 56.6605,Z 77,A 47.421,B 24.8792,C -2.5364,E1 25.0954,E2 396.8235} C_DIS
LIN {X 43.2956,Y 55.0656,Z 77,A 44.7717,B 24.8808,C -2.5198,E1 25.1013,E2 399.5022} C_DIS
LIN {X 46.1416,Y 52.7035,Z 77,A 42.0911,B 24.8805,C -2.523,E1 25.1069,E2 402.1646} C_DIS
LIN {X 48.9934,Y 50.0646,Z 77,A 39.36,B 24.88,C -2.5284,E1 25.1124,E2 404.8718} C_DIS
LIN {X 50.2503,Y 48.8025,Z 77,A 37.642,B 24.8809,C -2.5184,E1 25.1158,E2 406.6062} C_DIS
LIN {X 52.3296,Y 46.5657,Z 77,A 35.0629,B 24.8817,C -2.5107,E1 25.1207,E2 409.1921} C_DIS
LIN {X 53.9301,Y 44.7018,Z 77,A 32.6466,B 24.8831,C -2.4952,E1 25.1251,E2 411.6338} C_DIS
LIN {X 56.2399,Y 41.7604,Z 77,A 29.9173,B 24.883,C -2.4967,E1 25.1296,E2 414.3468} C_DIS
LIN {X 58.5789,Y 38.4089,Z 77,A 27.2278,B 24.8821,C -2.506,E1 25.1338,E2 417.001} C_DIS
LIN {X 60.1033,Y 35.9768,Z 77,A 24.023,B 24.8849,C -2.4767,E1 25.1386,E2 420.2588} C_DIS
LIN {X 62.0877,Y 32.4326,Z 77,A 21.3918,B 24.884,C -2.4865,E1 25.1421,E2 422.8529} C_DIS
LIN {X 63.9015,Y 28.6935,Z 77,A 17.989,B 24.8848,C -2.477,E1 25.1462,E2 426.26} C_DIS
LIN {X 65.5393,Y 24.7247,Z 77,A 14.5569,B 24.8856,C -2.4691,E1 25.1498,E2 429.6918} C_DIS
LIN {X 66.2608,Y 22.7185,Z 77,A 11.7585,B 24.8887,C -2.4352,E1 25.1524,E2 432.5547} C_DIS
LIN {X 67.3047,Y 19.4137,Z 77,A 9.6479,B 24.8877,C -2.4465,E1 25.154,E2 434.6264} C_DIS
LIN {X 68.0582,Y 16.5764,Z 77,A 7.0238,B 24.8889,C -2.4331,E1 25.1558,E2 437.2671} C_DIS
LIN {X 69.0722,Y 11.6508,Z 77,A 3.2958,B 24.8891,C -2.4311,E1 25.1578,E2 440.978} C_DIS
LIN {X 69.4927,Y 8.804,Z 77,A 1.0694,B 24.8894,C -2.4273,E1 25.1586,E2 443.2003} C_DIS
LIN {X 69.8631,Y 5.0973,Z 77,A -2.5308,B 24.8917,C -2.4024,E1 25.1595,E2 446.8379} C_DIS
LIN {X 70.0403,Y 1.0571,Z 77,A -5.5126,B 24.8918,C -2.4009,E1 25.1598,E2 449.8055} C_DIS
LIN {X 70.0074,Y -2.3942,Z 77,A -8.9323,B 24.8941,C -2.3755,E1 25.1595,E2 453.2648} C_DIS
LIN {X 69.8188,Y -5.6611,Z 77,A -10.2668,B 24.8915,C -2.4043,E1 25.1593,E2 454.5236} C_DIS
LIN {X 69.4038,Y -9.4844,Z 77,A -14.0785,B 24.8941,C -2.3756,E1 25.1581,E2 458.3803} C_DIS
LIN {X 68.9156,Y -12.5442,Z 77,A -16.5663,B 24.8947,C -2.3689,E1 25.1569,E2 460.8694} C_DIS
LIN {X 68.4526,Y -14.8643,Z 77,A -18.7701,B 24.8959,C -2.3554,E1 25.1556,E2 463.0924} C_DIS
LIN {X 67.4381,Y -18.9427,Z 77,A -21.6878,B 24.8956,C -2.359,E1 25.1536,E2 465.9846} C_DIS
LIN {X 66.5126,Y -21.9754,Z 77,A -24.7239,B 24.8974,C -2.3387,E1 25.151,E2 469.0514} C_DIS
LIN {X 64.69,Y -26.8708,Z 77,A -28.7279,B 24.8979,C -2.3332,E1 25.1469,E2 473.0463} C_DIS
LIN {X 63.5147,Y -29.5394,Z 77,A -31.5737,B 24.8996,C -2.3134,E1 25.1436,E2 475.9233} C_DIS
LIN {X 61.9333,Y -32.7259,Z 77,A -34.8602,B 24.9012,C -2.2947,E1 25.1393,E2 479.2369} C_DIS
LIN {X 60.0327,Y -36.0955,Z 77,A -37.1431,B 24.8999,C -2.3097,E1 25.1361,E2 481.4725} C_DIS
LIN {X 58.0227,Y -39.2435,Z 77,A -40.1581,B 24.9005,C -2.3023,E1 25.1315,E2 484.4899} C_DIS
LIN {X 56.3087,Y -41.6672,Z 77,A -42.6007,B 24.9012,C -2.2953,E1 25.1275,E2 486.9371} C_DIS
LIN {X 54.6689,Y -43.7969,Z 77,A -45.0611,B 24.9023,C -2.2824,E1 25.1232,E2 489.4166} C_DIS
LIN {X 51.3129,Y -47.685,Z 77,A -48.9755,B 24.9025,C -2.2796,E1 25.116,E2 493.3201} C_DIS
LIN {X 49.1352,Y -49.9244,Z 77,A -51.5048,B 24.903,C -2.2742,E1 25.111,E2 495.8515} C_DIS
LIN {X 45.9282,Y -52.8899,Z 77,A -55.4006,B 24.9044,C -2.2573,E1 25.1028,E2 499.7716} C_DIS
LIN {X 42.7624,Y -55.4804,Z 77,A -58.1872,B 24.9037,C -2.2651,E1 25.0968,E2 502.5293} C_DIS
LIN {X 39.6713,Y -57.7319,Z 77,A -61.2496,B 24.9041,C -2.2605,E1 25.0899,E2 505.5919} C_DIS
LIN {X 37.0318,Y -59.4589,Z 77,A -64.1162,B 24.9052,C -2.2479,E1 25.0831,E2 508.479} C_DIS
LIN {X 32.245,Y -62.1863,Z 77,A -68.2592,B 24.9051,C -2.2496,E1 25.073,E2 512.6057} C_DIS
LIN {X 28.4667,Y -64.0036,Z 77,A -71.9833,B 24.9062,C -2.2366,E1 25.0636,E2 516.3512} C_DIS
LIN {X 26.3893,Y -64.8869,Z 77,A -74.2049,B 24.9072,C -2.2242,E1 25.0578,E2 518.5969} C_DIS
LIN {X 21.8283,Y -66.5604,Z 77,A -78.042,B 24.9073,C -2.2227,E1 25.0476,E2 522.4299} C_DIS
LIN {X 18.7104,Y -67.5039,Z 77,A -81.3606,B 24.9089,C -2.2032,E1 25.0386,E2 525.7894} C_DIS
LIN {X 14.8715,Y -68.451,Z 77,A -83.6275,B 24.9072,C -2.2247,E1 25.0326,E2 528.0021} C_DIS
LIN {X 11.8981,Y -69.0309,Z 77,A -86.1336,B 24.9074,C -2.222,E1 25.0257,E2 530.5118} C_DIS
LIN {X 9.0379,Y -69.4624,Z 77,A -89.2878,B 24.9092,C -2.2007,E1 25.0168,E2 533.7139} C_DIS
LIN {X 5.4126,Y -69.8386,Z 77,A -91.1449,B 24.9069,C -2.2273,E1 25.0119,E2 535.5069} C_DIS
LIN {X 1.5463,Y -70.0313,Z 77,A -94.589,B 24.9076,C -2.2192,E1 25.0022,E2 538.9692} C_DIS
LIN {X 1.5463,Y -70.0313,Z 77,A -94.589,B 24.9076,C -2.2192,E1 25.0022,E2 538.9692} C_DIS
Enddeposition()
LIN {X 0.4437,Y -69.0924,Z 77,A -94.8738,B 24.9049,C -2.251,E1 25.0016,E2 539.1786} C_DIS
Startdeposition()
$VEL.CP = VEL_PRINT
LIN {X 2.6509,Y -69.0454,Z 77,A -92.2761,B 24.9033,C -2.2708,E1 25.009,E2 536.5346} C_DIS
LIN {X 5.8007,Y -68.8523,Z 77,A -89.5379,B 24.9029,C -2.2751,E1 25.0166,E2 533.7875} C_DIS
LIN {X 9.171,Y -68.4849,Z 77,A -87.1017,B 24.9036,C -2.2673,E1 25.0233,E2 531.3717} C_DIS
LIN {X 12.1187,Y -68.0247,Z 77,A -84.7482,B 24.9036,C -2.266,E1 25.0298,E2 529.0235} C_DIS
LIN {X 14.6832,Y -67.5175,Z 77,A -81.5752,B 24.9013,C -2.294,E1 25.0386,E2 525.7883} C_DIS
LIN {X 18.4474,Y -66.5888,Z 77,A -79.3663,B 24.9032,C -2.2711,E1 25.0444,E2 523.6372} C_DIS
LIN {X 21.1021,Y -65.7947,Z 77,A -76.2587,B 24.9012,C -2.295,E1 25.0528,E2 520.4787} C_DIS
LIN {X 24.2843,Y -64.6879,Z 77,A -74.6312,B 24.9035,C -2.2681,E1 25.0569,E2 518.9184} C_DIS
LIN {X 27.2601,Y -63.492,Z 77,A -71.5251,B 24.9022,C -2.2835,E1 25.065,E2 515.7829} C_DIS
LIN {X 30.0892,Y -62.2003,Z 77,A -68.9434,B 24.9018,C -2.2876,E1 25.0715,E2 513.1981} C_DIS
LIN {X 35.3646,Y -59.36,Z 77,A -64.2125,B 24.9016,C -2.2899,E1 25.0831,E2 508.4756} C_DIS
LIN {X 37.518,Y -58.0229,Z 77,A -61.4609,B 24.8998,C -2.3113,E1 25.0897,E2 505.6822} C_DIS
LIN {X 41.233,Y -55.445,Z 77,A -58.5277,B 24.901,C -2.2969,E1 25.0962,E2 502.7933} C_DIS
LIN {X 42.8148,Y -54.2319,Z 77,A -56.5776,B 24.9,C -2.3084,E1 25.1006,E2 500.8232} C_DIS
LIN {X 45.3516,Y -52.1292,Z 77,A -53.6435,B 24.899,C -2.32,E1 25.1068,E2 497.8731} C_DIS
LIN {X 47.9835,Y -49.7171,Z 77,A -50.9291,B 24.899,C -2.3202,E1 25.1123,E2 495.1693} C_DIS
LIN {X 50.1344,Y -47.5482,Z 77,A -48.335,B 24.8983,C -2.328,E1 25.1174,E2 492.5679} C_DIS
LIN {X 52.6298,Y -44.7696,Z 77,A -45.2893,B 24.8977,C -2.3345,E1 25.123,E2 489.5205} C_DIS
LIN {X 54.1199,Y -42.9566,Z 77,A -43.4046,B 24.8974,C -2.3379,E1 25.1263,E2 487.6366} C_DIS
LIN {X 56.0091,Y -40.4642,Z 77,A -40.8597,B 24.897,C -2.3435,E1 25.1305,E2 485.0907} C_DIS
LIN {X 57.8003,Y -37.8584,Z 77,A -38.2699,B 24.8964,C -2.3499,E1 25.1346,E2 482.4987} C_DIS
LIN {X 59.0455,Y -35.8863,Z 77,A -35.0936,B 24.8928,C -2.39,E1 25.1393,E2 479.2438} C_DIS
LIN {X 61.256,Y -31.9683,Z 77,A -32.9091,B 24.8957,C -2.3576,E1 25.1421,E2 477.1472} C_DIS
LIN {X 62.8223,Y -28.77,Z 77,A -29.7736,B 24.8945,C -2.3714,E1 25.1459,E2 473.996} C_DIS
LIN {X 63.8536,Y -26.4021,Z 77,A -27.486,B 24.8935,C -2.3819,E1 25.1484,E2 471.6962} C_DIS
LIN {X 64.8605,Y -23.819,Z 77,A -24.6736,B 24.8916,C -2.4033,E1 25.1512,E2 468.849} C_DIS
LIN {X 66.2248,Y -19.7101,Z 77,A -22.0206,B 24.893,C -2.3882,E1 25.1534,E2 466.2467} C_DIS
LIN {X 66.874,Y -17.3814,Z 77,A -19.4005,B 24.8909,C -2.4116,E1 25.1553,E2 463.5863} C_DIS
LIN {X 67.5646,Y -14.4673,Z 77,A -17.1782,B 24.8909,C -2.4121,E1 25.1566,E2 461.3757} C_DIS
LIN {X 68.1361,Y -11.4754,Z 77,A -14.7281,B 24.8903,C -2.418,E1 25.1578,E2 458.9261} C_DIS
LIN {X 68.562,Y -8.5764,Z 77,A -11.8886,B 24.8885,C -2.4371,E1 25.1589,E2 456.058} C_DIS
LIN {X 68.8571,Y -5.7415,Z 77,A -9.6136,B 24.8881,C -2.4422,E1 25.1594,E2 453.7847} C_DIS
LIN {X 69.0481,Y -2.5889,Z 77,A -7.2587,B 24.888,C -2.4431,E1 25.1597,E2 451.4416} C_DIS
LIN {X 69.0934,Y 0.554,Z 77,A -4.8573,B 24.8877,C -2.4456,E1 25.1597,E2 449.0484} C_DIS
LIN {X 69.0139,Y 3.3866,Z 77,A -2.3197,B 24.8866,C -2.4583,E1 25.1595,E2 446.496} C_DIS
LIN {X 68.7604,Y 6.8089,Z 77,A 0.2899,B 24.8864,C -2.4607,E1 25.1589,E2 443.8964} C_DIS
LIN {X 68.4699,Y 9.2871,Z 77,A 2.5197,B 24.8853,C -2.4716,E1 25.1581,E2 441.6538} C_DIS
LIN {X 67.9833,Y 12.3487,Z 77,A 5.1982,B 24.8843,C -2.4826,E1 25.1568,E2 438.9652} C_DIS
LIN {X 67.2786,Y 15.7428,Z 77,A 7.6627,B 24.8846,C -2.48,E1 25.1553,E2 436.5212} C_DIS
LIN {X 66.6281,Y 18.3026,Z 77,A 9.9907,B 24.8836,C -2.4904,E1 25.1537,E2 434.1819} C_DIS
LIN {X 64.9044,Y 23.6988,Z 77,A 14.5293,B 24.8827,C -2.4998,E1 25.1498,E2 429.6467} C_DIS
LIN {X 63.6302,Y 26.9336,Z 77,A 17.8743,B 24.8807,C -2.5207,E1 25.1462,E2 426.2707} C_DIS
LIN {X 62.2845,Y 29.9141,Z 77,A 20.1729,B 24.8811,C -2.5169,E1 25.1435,E2 423.9935} C_DIS
LIN {X 61.2726,Y 31.9368,Z 77,A 22.129,B 24.8804,C -2.5243,E1 25.141,E2 422.0304} C_DIS
LIN {X 59.922,Y 34.403,Z 77,A 25.2957,B 24.8776,C -2.5534,E1 25.1365,E2 418.8113} C_DIS
LIN {X 58.0543,Y 37.4691,Z 77,A 27.2212,B 24.8796,C -2.5323,E1 25.1338,E2 416.9454} C_DIS
LIN {X 55.5569,Y 41.0821,Z 77,A 31.245,B 24.8778,C -2.5516,E1 25.1272,E2 412.8955} C_DIS
LIN {X 53.2518,Y 44.0282,Z 77,A 34.1008,B 24.8778,C -2.5522,E1 25.1222,E2 410.0515} C_DIS
LIN {X 51.2262,Y 46.3705,Z 77,A 36.7243,B 24.877,C -2.5594,E1 25.1174,E2 407.4227} C_DIS
LIN {X 48.4974,Y 49.216,Z 77,A 39.7116,B 24.877,C -2.5589,E1 25.1116,E2 404.4495} C_DIS
LIN {X 45.4741,Y 52.0222,Z 77,A 43.5341,B 24.8754,C -2.5763,E1 25.1036,E2 400.6012} C_DIS
LIN {X 42.4336,Y 54.5317,Z 77,A 46.6163,B 24.8753,C -2.5774,E1 25.0969,E2 397.5281} C_DIS
LIN {X 39.9558,Y 56.3718,Z 77,A 49.0026,B 24.8753,C -2.5772,E1 25.0916,E2 395.1507} C_DIS
LIN {X 36.3543,Y 58.7593,Z 77,A 53.2529,B 24.8731,C -2.6001,E1 25.0815,E2 390.8597} C_DIS
LIN {X 31.284,Y 61.608,Z 77,A 57.5736,B 24.8737,C -2.5935,E1 25.071,E2 386.5672} C_DIS
LIN {X 28.5479,Y 62.9226,Z 77,A 60.0134,B 24.8737,C -2.5945,E1 25.0648,E2 384.1313} C_DIS
LIN {X 25.4218,Y 64.2492,Z 77,A 63.5527,B 24.8715,C -2.6158,E1 25.0555,E2 380.5495} C_DIS
LIN {X 22.3712,Y 65.3746,Z 77,A 65.2239,B 24.8739,C -2.5921,E1 25.0513,E2 378.9379} C_DIS
LIN {X 18.9764,Y 66.4389,Z 77,A 68.8222,B 24.872,C -2.6106,E1 25.0416,E2 375.3021} C_DIS
LIN {X 15.0952,Y 67.4276,Z 77,A 71.7487,B 24.8728,C -2.6025,E1 25.0337,E2 372.399} C_DIS
LIN {X 12.7217,Y 67.9153,Z 77,A 74.0277,B 24.8721,C -2.61,E1 25.0274,E2 370.1048} C_DIS
LIN {X 9.2879,Y 68.4698,Z 77,A 76.77,B 24.8724,C -2.6073,E1 25.0198,E2 367.3715} C_DIS
LIN {X 6.4101,Y 68.7977,Z 77,A 79.1418,B 24.8724,C -2.6069,E1 25.0133,E2 365.0023} C_DIS
LIN {X 3.3205,Y 69.0167,Z 77,A 81.8323,B 24.8721,C -2.6098,E1 25.0057,E2 362.3057} C_DIS
LIN {X 0.047,Y 69.0966,Z 77,A 84.4739,B 24.8723,C -2.6076,E1 24.9984,E2 359.6698} C_DIS
LIN {X -3.3529,Y 69.0153,Z 77,A 87.3128,B 24.8723,C -2.6072,E1 24.9905,E2 356.8313} C_DIS
LIN {X -6.3382,Y 68.8043,Z 77,A 89.9403,B 24.8721,C -2.6095,E1 24.9831,E2 354.197} C_DIS
LIN {X -10.4371,Y 68.3029,Z 77,A 92.7705,B 24.8737,C -2.5934,E1 24.9754,E2 351.4032} C_DIS
LIN {X -12.7926,Y 67.9016,Z 77,A 95.2957,B 24.8726,C -2.6047,E1 24.9684,E2 348.8484} C_DIS
LIN {X -16.3042,Y 67.1445,Z 77,A 98.2167,B 24.873,C -2.6006,E1 24.9604,E2 345.9333} C_DIS
LIN {X -19.7461,Y 66.214,Z 77,A 101.0196,B 24.8737,C -2.594,E1 24.9529,E2 343.1418} C_DIS
LIN {X -22.0815,Y 65.4722,Z 77,A 103.0261,B 24.874,C -2.591,E1 24.9476,E2 341.1386} C_DIS
LIN {X -25.506,Y 64.2162,Z 77,A 106.2057,B 24.874,C -2.5906,E1 24.9393,E2 337.9534} C_DIS
LIN {X -29.4437,Y 62.509,Z 77,A 109.4673,B 24.8752,C -2.5786,E1 24.931,E2 334.7126} C_DIS
LIN {X -31.286,Y 61.607,Z 77,A 111.4315,B 24.8749,C -2.5818,E1 24.9261,E2 332.7353} C_DIS
LIN {X -34.0595,Y 60.1193,Z 77,A 114.738,B 24.8737,C -2.5932,E1 24.918,E2 329.3921} C_DIS
LIN {X -36.8257,Y 58.4649,Z 77,A 116.7211,B 24.8757,C -2.5727,E1 24.9134,E2 327.4518} C_DIS
LIN {X -39.2303,Y 56.8793,Z 77,A 119.5895,B 24.8751,C -2.5788,E1 24.9067,E2 324.559} C_DIS
LIN {X -41.8198,Y 55.0043,Z 77,A 122.1295,B 24.8759,C -2.5708,E1 24.901,E2 322.029} C_DIS
LIN {X -45.5859,Y 51.9246,Z 77,A 125.526,B 24.8781,C -2.5479,E1 24.8939,E2 318.6742} C_DIS
LIN {X -48.1479,Y 49.5566,Z 77,A 128.9868,B 24.8776,C -2.5537,E1 24.8868,E2 315.1854} C_DIS
LIN {X -51.2082,Y 46.3876,Z 77,A 132.9939,B 24.8776,C -2.5525,E1 24.8791,E2 311.1635} C_DIS
LIN {X -54.7645,Y 42.1314,Z 77,A 137.4389,B 24.8792,C -2.5372,E1 24.8714,E2 306.7343} C_DIS
LIN {X -56.7074,Y 39.4776,Z 77,A 140.7038,B 24.8787,C -2.5415,E1 24.8661,E2 303.443} C_DIS
LIN {X -58.807,Y 36.278,Z 77,A 142.6867,B 24.882,C -2.5069,E1 24.8633,E2 301.5328} C_DIS
LIN {X -60.4059,Y 33.5463,Z 77,A 145.6282,B 24.882,C -2.5062,E1 24.8592,E2 298.5775} C_DIS
LIN {X -62.3281,Y 29.8234,Z 77,A 149.2321,B 24.8828,C -2.4988,E1 24.8547,E2 294.9719} C_DIS
LIN {X -63.4999,Y 27.242,Z 77,A 151.5724,B 24.8835,C -2.4916,E1 24.852,E2 292.6361} C_DIS
LIN {X -64.6941,Y 24.2679,Z 77,A 155.1199,B 24.8824,C -2.5027,E1 24.8485,E2 289.042} C_DIS
LIN {X -65.9544,Y 20.597,Z 77,A 157.4255,B 24.8852,C -2.4732,E1 24.8466,E2 286.7938} C_DIS
LIN {X -67.1759,Y 16.1726,Z 77,A 161.5227,B 24.8857,C -2.4675,E1 24.8437,E2 282.6862} C_DIS
LIN {X -68.2209,Y 10.9672,Z 77,A 166.2769,B 24.8863,C -2.4611,E1 24.8413,E2 277.9191} C_DIS
LIN {X -68.6593,Y 7.7575,Z 77,A 168.7933,B 24.8874,C -2.4489,E1 24.8405,E2 275.4167} C_DIS
LIN {X -69.0106,Y 3.4458,Z 77,A 171.9704,B 24.8893,C -2.4288,E1 24.8399,E2 272.2686} C_DIS
LIN {X -69.0926,Y 0.7029,Z 77,A 174.4183,B 24.8896,C -2.4253,E1 24.8398,E2 269.8145} C_DIS
LIN {X -69.0167,Y -3.3216,Z 77,A 177.4074,B 24.8912,C -2.4073,E1 24.84,E2 266.8503} C_DIS
LIN {X -68.9025,Y -5.1737,Z 77,A 179.1442,B 24.8913,C -2.4067,E1 24.8404,E2 265.1045} C_DIS
LIN {X -68.6577,Y -7.7716,Z 77,A -178.7241,B 24.892,C -2.3992,E1 24.841,E2 262.9779} C_DIS
LIN {X -68.3299,Y -10.2623,Z 77,A -176.2856,B 24.8919,C -2.4003,E1 24.842,E2 260.5222} C_DIS
LIN {X -67.8875,Y -12.8659,Z 77,A -173.3092,B 24.8909,C -2.4106,E1 24.8436,E2 257.5036} C_DIS
LIN {X -67.0162,Y -16.8279,Z 77,A -171.2085,B 24.8943,C -2.3731,E1 24.8449,E2 255.4801} C_DIS
LIN {X -65.8135,Y -21.044,Z 77,A -167.3224,B 24.8948,C -2.3676,E1 24.8479,E2 251.5847} C_DIS
LIN {X -64.9182,Y -23.6608,Z 77,A -164.931,B 24.8952,C -2.3631,E1 24.8502,E2 249.1906} C_DIS
LIN {X -63.4796,Y -27.2887,Z 77,A -161.7093,B 24.8961,C -2.3535,E1 24.8536,E2 245.9738} C_DIS
LIN {X -62.326,Y -29.8276,Z 77,A -159.3298,B 24.8965,C -2.3486,E1 24.8564,E2 243.5932} C_DIS
LIN {X -60.196,Y -33.9215,Z 77,A -155.3953,B 24.8972,C -2.3406,E1 24.8616,E2 239.6568} C_DIS
LIN {X -58.3478,Y -37.0118,Z 77,A -152.4862,B 24.898,C -2.3312,E1 24.8658,E2 236.7553} C_DIS
LIN {X -55.9061,Y -40.6051,Z 77,A -148.8006,B 24.8987,C -2.3241,E1 24.8717,E2 233.0685} C_DIS
LIN {X -53.9354,Y -43.1896,Z 77,A -146.1241,B 24.8992,C -2.3173,E1 24.8763,E2 230.3955} C_DIS
LIN {X -51.2467,Y -46.3477,Z 77,A -143.033,B 24.9006,C -2.3018,E1 24.8819,E2 227.3274} C_DIS
LIN {X -48.8582,Y -48.8596,Z 77,A -139.7121,B 24.9003,C -2.3058,E1 24.8884,E2 223.9829} C_DIS
LIN {X -45.8603,Y -51.6822,Z 77,A -136.2646,B 24.9008,C -2.2998,E1 24.8955,E2 220.5357} C_DIS
LIN {X -43.2627,Y -53.8762,Z 77,A -133.51,B 24.9013,C -2.2931,E1 24.9014,E2 217.7866} C_DIS
LIN {X -39.723,Y -56.5368,Z 77,A -130.1085,B 24.9024,C -2.2806,E1 24.9091,E2 214.4028} C_DIS
LIN {X -37.8,Y -57.8398,Z 77,A -126.8758,B 24.9,C -2.3081,E1 24.9168,E2 211.0941} C_DIS
LIN {X -34.1813,Y -60.0494,Z 77,A -124.7461,B 24.9033,C -2.2707,E1 24.9217,E2 209.0472} C_DIS
LIN {X -32.3002,Y -61.0812,Z 77,A -122.6606,B 24.9029,C -2.2755,E1 24.9269,E2 206.9443} C_DIS
LIN {X -29.4977,Y -62.4839,Z 77,A -120.0448,B 24.9031,C -2.2728,E1 24.9335,E2 204.3281} C_DIS
LIN {X -25.3979,Y -64.2587,Z 77,A -116.5499,B 24.9038,C -2.264,E1 24.9424,E2 200.846} C_DIS
LIN {X -22.059,Y -65.4798,Z 77,A -113.0124,B 24.9028,C -2.2757,E1 24.9518,E2 197.274} C_DIS
LIN {X -18.6407,Y -66.534,Z 77,A -110.3676,B 24.9037,C -2.2659,E1 24.9589,E2 194.648} C_DIS
LIN {X -15.8483,Y -67.2542,Z 77,A -107.8421,B 24.9035,C -2.2679,E1 24.9657,E2 192.1142} C_DIS
LIN {X -11.9596,Y -68.0533,Z 77,A -104.8378,B 24.9042,C -2.2596,E1 24.9739,E2 189.1263} C_DIS
LIN {X -9.2394,Y -68.4761,Z 77,A -102.4597,B 24.9041,C -2.2614,E1 24.9805,E2 186.742} C_DIS
LIN {X -6.3494,Y -68.8033,Z 77,A -99.7989,B 24.9036,C -2.2674,E1 24.988,E2 184.0656} C_DIS
LIN {X -2.5871,Y -69.0482,Z 77,A -97.1321,B 24.9045,C -2.2561,E1 24.9953,E2 181.4247} C_DIS
LIN {X -0.0674,Y -69.0965,Z 77,A -94.8957,B 24.9042,C -2.2602,E1 25.0016,E2 179.1786} C_DIS
LIN {X -0.0674,Y -69.0965,Z 77,A -94.8957,B 24.9042,C -2.2602,E1 25.0016,E2 179.1786} C_DIS
Enddeposition()
LIN {X 0.4295,Y -68.141,Z 77,A -94.5394,B 24.9029,C -2.2753,E1 25.0027,E2 178.7864} C_DIS
Startdeposition()
$VEL.CP = VEL_PRINT
LIN {X -2.6329,Y -68.0932,Z 77,A -98.0429,B 24.9048,C -2.2522,E1 24.9928,E2 182.3449} C_DIS
LIN {X -5.3064,Y -67.9366,Z 77,A -100.431,B 24.9051,C -2.249,E1 24.9861,E2 184.7417} C_DIS
LIN {X -8.1788,Y -67.6513,Z 77,A -102.8112,B 24.905,C -2.2504,E1 24.9795,E2 187.12} C_DIS
LIN {X -10.7451,Y -67.2917,Z 77,A -105.049,B 24.905,C -2.2495,E1 24.9733,E2 189.3618} C_DIS
LIN {X -13.5687,Y -66.779,Z 77,A -107.4378,B 24.905,C -2.251,E1 24.9667,E2 191.7497} C_DIS
LIN {X -16.4085,Y -66.1389,Z 77,A -109.8292,B 24.9047,C -2.2535,E1 24.9602,E2 194.1383} C_DIS
LIN {X -19.0062,Y -65.4404,Z 77,A -111.8773,B 24.9042,C -2.2599,E1 24.9548,E2 196.1743} C_DIS
LIN {X -22.0811,Y -64.4675,Z 77,A -114.8193,B 24.9045,C -2.2566,E1 24.9469,E2 199.1294} C_DIS
LIN {X -24.6855,Y -63.5154,Z 77,A -117.1327,B 24.9043,C -2.2592,E1 24.9409,E2 201.4417} C_DIS
LIN {X -27.2928,Y -62.439,Z 77,A -119.5647,B 24.9042,C -2.2602,E1 24.9346,E2 203.8768} C_DIS
LIN {X -29.9174,Y -61.226,Z 77,A -122.1311,B 24.9042,C -2.26,E1 24.9281,E2 206.4503} C_DIS
LIN {X -32.8221,Y -59.7191,Z 77,A -124.7757,B 24.9037,C -2.2659,E1 24.9216,E2 209.0881} C_DIS
LIN {X -35.8703,Y -57.939,Z 77,A -127.7627,B 24.9033,C -2.2698,E1 24.9145,E2 212.0751} C_DIS
LIN {X -38.5563,Y -56.1881,Z 77,A -130.581,B 24.9033,C -2.2713,E1 24.9079,E2 214.8992} C_DIS
LIN {X -41.3302,Y -54.1797,Z 77,A -133.3821,B 24.9026,C -2.2779,E1 24.9016,E2 217.6944} C_DIS
LIN {X -43.912,Y -52.1094,Z 77,A -136.0155,B 24.9019,C -2.2863,E1 24.896,E2 220.3178} C_DIS
LIN {X -46.2827,Y -50.0151,Z 77,A -138.8718,B 24.9019,C -2.2872,E1 24.89,E2 223.1833} C_DIS
LIN {X -48.4037,Y -47.9648,Z 77,A -141.2832,B 24.9013,C -2.2939,E1 24.8853,E2 225.589} C_DIS
LIN {X -50.5084,Y -45.7447,Z 77,A -143.9119,B 24.9009,C -2.2982,E1 24.8803,E2 228.2189} C_DIS
LIN {X -52.292,Y -43.6933,Z 77,A -146.2504,B 24.9006,C -2.3023,E1 24.876,E2 230.5583} C_DIS
LIN {X -54.1756,Y -41.3356,Z 77,A -148.6684,B 24.8998,C -2.3108,E1 24.8719,E2 232.9674} C_DIS
LIN {X -55.7823,Y -39.1402,Z 77,A -151.1668,B 24.8998,C -2.3119,E1 24.8678,E2 235.4754} C_DIS
LIN {X -57.4801,Y -36.6008,Z 77,A -153.5335,B 24.8988,C -2.3227,E1 24.8642,E2 237.8282} C_DIS
LIN {X -58.6988,Y -34.6119,Z 77,A -156.0658,B 24.8994,C -2.3159,E1 24.8606,E2 240.39} C_DIS
LIN {X -60.8794,Y -30.6166,Z 77,A -159.4963,B 24.8977,C -2.3344,E1 24.8561,E2 243.7943} C_DIS
LIN {X -62.1988,Y -27.8363,Z 77,A -161.7661,B 24.8965,C -2.3483,E1 24.8535,E2 246.0434} C_DIS
LIN {X -62.9525,Y -26.0886,Z 77,A -163.774,B 24.8969,C -2.3443,E1 24.8513,E2 248.0719} C_DIS
LIN {X -64.0401,Y -23.2894,Z 77,A -166.0954,B 24.8959,C -2.3559,E1 24.849,E2 250.3789} C_DIS
LIN {X -64.8648,Y -20.8827,Z 77,A -168.0278,B 24.8949,C -2.3664,E1 24.8473,E2 252.2971} C_DIS
LIN {X -65.7114,Y -18.0447,Z 77,A -170.8545,B 24.8949,C -2.3669,E1 24.8451,E2 255.1391} C_DIS
LIN {X -66.4324,Y -15.1753,Z 77,A -173.0923,B 24.8937,C -2.3796,E1 24.8436,E2 257.3596} C_DIS
LIN {X -67.0978,Y -11.8929,Z 77,A -176.2083,B 24.8935,C -2.382,E1 24.842,E2 260.4882} C_DIS
LIN {X -67.5587,Y -8.9088,Z 77,A -178.6836,B 24.8927,C -2.3912,E1 24.841,E2 262.9563} C_DIS
LIN {X -67.8771,Y -6.0232,Z 77,A 178.7674,B 24.8922,C -2.3966,E1 24.8403,E2 265.5077} C_DIS
LIN {X -68.0391,Y -3.7684,Z 77,A 176.9144,B 24.8916,C -2.4036,E1 24.84,E2 267.3551} C_DIS
LIN {X -68.1309,Y -1.3039,Z 77,A 174.9892,B 24.8907,C -2.4132,E1 24.8398,E2 269.269} C_DIS
LIN {X -68.128,Y 1.4658,Z 77,A 172.3199,B 24.8907,C -2.4136,E1 24.8398,E2 271.9534} C_DIS
LIN {X -67.9439,Y 5.2149,Z 77,A 169.26,B 24.8896,C -2.4256,E1 24.8404,E2 275.0031} C_DIS
LIN {X -67.5965,Y 8.617,Z 77,A 165.4781,B 24.8904,C -2.4164,E1 24.8417,E2 278.8294} C_DIS
LIN {X -67.0393,Y 12.2183,Z 77,A 163.3152,B 24.8879,C -2.4442,E1 24.8427,E2 280.9387} C_DIS
LIN {X -66.6376,Y 14.249,Z 77,A 160.9961,B 24.8884,C -2.438,E1 24.844,E2 283.2865} C_DIS
LIN {X -65.6513,Y 18.2631,Z 77,A 157.9885,B 24.8866,C -2.4583,E1 24.8461,E2 286.2631} C_DIS
LIN {X -64.8035,Y 21.0722,Z 77,A 155.6094,B 24.8857,C -2.4677,E1 24.8481,E2 288.6334} C_DIS
LIN {X -63.7173,Y 24.1585,Z 77,A 152.696,B 24.8852,C -2.4727,E1 24.8509,E2 291.5511} C_DIS
LIN {X -62.6287,Y 26.8577,Z 77,A 150.3117,B 24.8844,C -2.4814,E1 24.8535,E2 293.9282} C_DIS
LIN {X -61.7376,Y 28.8444,Z 77,A 148.2352,B 24.8844,C -2.4818,E1 24.8559,E2 296.015} C_DIS
LIN {X -60.0865,Y 32.1448,Z 77,A 145.2574,B 24.8833,C -2.4933,E1 24.8597,E2 298.9811} C_DIS
LIN {X -58.4092,Y 35.0999,Z 77,A 142.5235,B 24.8823,C -2.504,E1 24.8635,E2 301.7037} C_DIS
LIN {X -56.7328,Y 37.7484,Z 77,A 139.3117,B 24.8827,C -2.4994,E1 24.8685,E2 304.9426} C_DIS
LIN {X -54.0103,Y 41.5502,Z 77,A 135.8263,B 24.8809,C -2.5191,E1 24.8742,E2 308.3978} C_DIS
LIN {X -52.2098,Y 43.7922,Z 77,A 132.4573,B 24.8822,C -2.5056,E1 24.8803,E2 311.8146} C_DIS
LIN {X -49.6739,Y 46.6479,Z 77,A 130.3157,B 24.8793,C -2.5357,E1 24.8843,E2 313.8937} C_DIS
LIN {X -46.5399,Y 49.7755,Z 77,A 126.391,B 24.8789,C -2.5402,E1 24.8921,E2 317.8241} C_DIS
LIN {X -44.9463,Y 51.2189,Z 77,A 123.9939,B 24.8797,C -2.5319,E1 24.8972,E2 320.2506} C_DIS
LIN {X -41.0833,Y 54.3666,Z 77,A 120.4094,B 24.8776,C -2.5535,E1 24.905,E2 323.7966} C_DIS
LIN {X -38.5234,Y 56.2105,Z 77,A 117.6629,B 24.8773,C -2.5568,E1 24.9112,E2 326.5448} C_DIS
LIN {X -35.7188,Y 58.0331,Z 77,A 114.6529,B 24.8772,C -2.5577,E1 24.9184,E2 329.562} C_DIS
LIN {X -32.5585,Y 59.8621,Z 77,A 111.9638,B 24.8759,C -2.5713,E1 24.9248,E2 332.2267} C_DIS
LIN {X -30.1663,Y 61.1026,Z 77,A 109.7498,B 24.8754,C -2.5761,E1 24.9303,E2 334.4352} C_DIS
LIN {X -27.9119,Y 62.1646,Z 77,A 107.4209,B 24.8756,C -2.5741,E1 24.9363,E2 336.7746} C_DIS
LIN {X -25.2126,Y 63.3084,Z 77,A 104.7759,B 24.8756,C -2.5735,E1 24.9431,E2 339.427} C_DIS
LIN {X -21.1034,Y 64.7934,Z 77,A 100.7135,B 24.8761,C -2.5694,E1 24.9539,E2 343.5069} C_DIS
LIN {X -15.6433,Y 66.3243,Z 77,A 96.7849,B 24.8738,C -2.593,E1 24.9644,E2 347.3853} C_DIS
LIN {X -13.1849,Y 66.8564,Z 77,A 94.3965,B 24.8742,C -2.5885,E1 24.9709,E2 349.7871} C_DIS
LIN {X -10.4321,Y 67.3401,Z 77,A 92.3728,B 24.8733,C -2.5977,E1 24.9765,E2 351.791} C_DIS
LIN {X -8.6839,Y 67.5879,Z 77,A 90.5508,B 24.874,C -2.5908,E1 24.9816,E2 353.6306} C_DIS
LIN {X -5.8201,Y 67.8955,Z 77,A 88.1331,B 24.8739,C -2.5921,E1 24.9883,E2 356.0465} C_DIS
LIN {X -2.9142,Y 68.0811,Z 77,A 85.8031,B 24.8735,C -2.5958,E1 24.9947,E2 358.3685} C_DIS
LIN {X -0.1362,Y 68.1439,Z 77,A 83.4272,B 24.8735,C -2.5954,E1 25.0014,E2 360.7454} C_DIS
LIN {X 2.7185,Y 68.0895,Z 77,A 81.0086,B 24.8735,C -2.5952,E1 25.0081,E2 363.1639} C_DIS
LIN {X 5.4482,Y 67.9253,Z 77,A 78.6438,B 24.8737,C -2.5936,E1 25.0147,E2 365.5315} C_DIS
LIN {X 8.2009,Y 67.6487,Z 77,A 76.3367,B 24.8737,C -2.5937,E1 25.0211,E2 367.8367} C_DIS
LIN {X 11.1402,Y 67.2267,Z 77,A 73.9395,B 24.8735,C -2.5954,E1 25.0277,E2 370.2277} C_DIS
LIN {X 13.7695,Y 66.7378,Z 77,A 71.6148,B 24.8738,C -2.5926,E1 25.0341,E2 372.5562} C_DIS
LIN {X 16.5234,Y 66.1109,Z 77,A 68.6718,B 24.8753,C -2.5776,E1 25.0422,E2 375.5305} C_DIS
LIN {X 20.6875,Y 64.928,Z 77,A 65.5977,B 24.8742,C -2.5887,E1 25.0503,E2 378.573} C_DIS
LIN {X 22.8836,Y 64.1871,Z 77,A 63.5568,B 24.8746,C -2.5847,E1 25.0557,E2 380.6191} C_DIS
LIN {X 25.8213,Y 63.0619,Z 77,A 61.1356,B 24.8743,C -2.5877,E1 25.062,E2 383.028} C_DIS
LIN {X 28.1198,Y 62.0711,Z 77,A 58.9007,B 24.8748,C -2.5821,E1 25.0677,E2 385.2706} C_DIS
LIN {X 30.6207,Y 60.8774,Z 77,A 56.8275,B 24.8745,C -2.5857,E1 25.0729,E2 387.3299} C_DIS
LIN {X 33.8485,Y 59.1424,Z 77,A 53.5291,B 24.8754,C -2.5761,E1 25.081,E2 390.6415} C_DIS
LIN {X 36.4291,Y 57.5898,Z 77,A 50.7235,B 24.8764,C -2.5654,E1 25.0877,E2 393.4634} C_DIS
LIN {X 39.2822,Y 55.6827,Z 77,A 48.0984,B 24.8763,C -2.5673,E1 25.0937,E2 396.0751} C_DIS
LIN {X 41.7236,Y 53.8767,Z 77,A 45.6644,B 24.8764,C -2.5659,E1 25.0991,E2 398.5037} C_DIS
LIN {X 44.8066,Y 51.3409,Z 77,A 42.1376,B 24.8774,C -2.5552,E1 25.1067,E2 402.0422} C_DIS
LIN {X 47.1792,Y 49.1698,Z 77,A 39.5945,B 24.8776,C -2.5539,E1 25.1118,E2 404.578} C_DIS
LIN {X 49.3118,Y 47.0319,Z 77,A 36.9651,B 24.8783,C -2.5461,E1 25.117,E2 407.2145} C_DIS
LIN {X 51.2453,Y 44.9162,Z 77,A 34.6196,B 24.8787,C -2.5425,E1 25.1213,E2 409.5582} C_DIS
LIN {X 53.1469,Y 42.6493,Z 77,A 31.5775,B 24.8806,C -2.5223,E1 25.1268,E2 412.6339} C_DIS
LIN {X 55.8113,Y 39.0984,Z 77,A 28.4339,B 24.88,C -2.5285,E1 25.1319,E2 415.7476} C_DIS
LIN {X 57.4331,Y 36.6741,Z 77,A 25.6552,B 24.8814,C -2.5137,E1 25.1361,E2 418.5474} C_DIS
LIN {X 59.2061,Y 33.7376,Z 77,A 23.1254,B 24.8812,C -2.5154,E1 25.1397,E2 421.0601} C_DIS
LIN {X 60.4575,Y 31.4411,Z 77,A 20.9387,B 24.8818,C -2.5098,E1 25.1426,E2 423.2486} C_DIS
LIN {X 61.5685,Y 29.2054,Z 77,A 18.0699,B 24.8842,C -2.4837,E1 25.1461,E2 426.1637} C_DIS
LIN {X 62.9464,Y 26.1042,Z 77,A 15.9445,B 24.8832,C -2.4948,E1 25.1483,E2 428.2512} C_DIS
LIN {X 64.0455,Y 23.2745,Z 77,A 13.5591,B 24.8834,C -2.4919,E1 25.1507,E2 430.6302} C_DIS
LIN {X 65.3284,Y 19.3835,Z 77,A 10.0858,B 24.8845,C -2.481,E1 25.1536,E2 434.1096} C_DIS
LIN {X 66.0372,Y 16.8118,Z 77,A 7.8347,B 24.8851,C -2.474,E1 25.1552,E2 436.3643} C_DIS
LIN {X 66.656,Y 14.1646,Z 77,A 5.6315,B 24.8856,C -2.4692,E1 25.1566,E2 438.5659} C_DIS
LIN {X 67.1237,Y 11.7488,Z 77,A 3.5489,B 24.8862,C -2.4625,E1 25.1576,E2 440.6522} C_DIS
LIN {X 67.5345,Y 9.0961,Z 77,A 1.0985,B 24.8873,C -2.4502,E1 25.1586,E2 443.1171} C_DIS
LIN {X 67.8898,Y 5.8856,Z 77,A -1.2248,B 24.8871,C -2.4523,E1 25.1593,E2 445.4217} C_DIS
LIN {X 68.0612,Y 3.3698,Z 77,A -3.6937,B 24.8886,C -2.4362,E1 25.1597,E2 447.914} C_DIS
LIN {X 68.1437,Y 0.0863,Z 77,A -6.3171,B 24.8891,C -2.4312,E1 25.1597,E2 450.5336} C_DIS
LIN {X 68.0933,Y -2.6299,Z 77,A -8.5879,B 24.8897,C -2.4243,E1 25.1596,E2 452.8073} C_DIS
LIN {X 67.8954,Y -5.8218,Z 77,A -11.4116,B 24.8908,C -2.4121,E1 25.159,E2 455.643} C_DIS
LIN {X 67.5657,Y -8.8546,Z 77,A -13.7774,B 24.8911,C -2.4094,E1 25.1582,E2 458.0013} C_DIS
LIN {X 67.1698,Y -11.4805,Z 77,A -15.9671,B 24.8916,C -2.4035,E1 25.1572,E2 460.1921} C_DIS
LIN {X 66.6751,Y -14.0745,Z 77,A -18.2221,B 24.8923,C -2.3955,E1 25.156,E2 462.4527} C_DIS
LIN {X 66.0982,Y -16.5746,Z 77,A -20.4774,B 24.8932,C -2.3861,E1 25.1545,E2 464.7172} C_DIS
LIN {X 65.282,Y -19.54,Z 77,A -22.6485,B 24.8929,C -2.3893,E1 25.1529,E2 466.8683} C_DIS
LIN {X 64.4391,Y -22.1652,Z 77,A -25.2833,B 24.8943,C -2.3736,E1 25.1505,E2 469.5254} C_DIS
LIN {X 63.2851,Y -25.2718,Z 77,A -28.0795,B 24.8951,C -2.3648,E1 25.1477,E2 472.3266} C_DIS
LIN {X 62.0692,Y -28.124,Z 77,A -30.4047,B 24.8951,C -2.3646,E1 25.1451,E2 474.6396} C_DIS
LIN {X 60.8021,Y -30.7686,Z 77,A -33.1606,B 24.8964,C -2.3496,E1 25.1417,E2 477.4164} C_DIS
LIN {X 59.1364,Y -33.8588,Z 77,A -36.2029,B 24.8974,C -2.3387,E1 25.1376,E2 480.4687} C_DIS
LIN {X 57.5747,Y -36.4533,Z 77,A -38.886,B 24.8983,C -2.3278,E1 25.1336,E2 483.1637} C_DIS
LIN {X 55.4307,Y -39.6354,Z 77,A -41.6714,B 24.8981,C -2.3308,E1 25.1292,E2 485.9285} C_DIS
LIN {X 53.7806,Y -41.8483,Z 77,A -44.0154,B 24.8987,C -2.324,E1 25.1252,E2 488.2775} C_DIS
LIN {X 52.0435,Y -43.9895,Z 77,A -46.369,B 24.8993,C -2.317,E1 25.121,E2 490.6366} C_DIS
LIN {X 50.069,Y -46.224,Z 77,A -48.8064,B 24.8997,C -2.3126,E1 25.1164,E2 493.0737} C_DIS
LIN {X 48.1206,Y -48.2498,Z 77,A -51.142,B 24.9001,C -2.3076,E1 25.1119,E2 495.4111} C_DIS
LIN {X 46.131,Y -50.1544,Z 77,A -53.2672,B 24.9001,C -2.3072,E1 25.1076,E2 497.5286} C_DIS
LIN {X 44.193,Y -51.8701,Z 77,A -55.6596,B 24.901,C -2.2966,E1 25.1025,E2 499.9365} C_DIS
LIN {X 41.7981,Y -53.8193,Z 77,A -58.1934,B 24.9014,C -2.2927,E1 25.0969,E2 502.4703} C_DIS
LIN {X 39.9021,Y -55.2404,Z 77,A -60.5294,B 24.9025,C -2.2796,E1 25.0916,E2 504.8289} C_DIS
LIN {X 36.0926,Y -57.8001,Z 77,A -63.861,B 24.902,C -2.2859,E1 25.0839,E2 508.1348} C_DIS
LIN {X 33.0534,Y -59.5906,Z 77,A -66.9606,B 24.9027,C -2.2771,E1 25.0764,E2 511.2457} C_DIS
LIN {X 30.53,Y -60.9224,Z 77,A -69.3382,B 24.903,C -2.2737,E1 25.0705,E2 513.6249} C_DIS
LIN {X 27.9529,Y -62.1463,Z 77,A -71.7246,B 24.9033,C -2.2703,E1 25.0644,E2 516.0131} C_DIS
LIN {X 25.1394,Y -63.3371,Z 77,A -74.2612,B 24.9035,C -2.2675,E1 25.0579,E2 518.5507} C_DIS
LIN {X 22.9053,Y -64.1795,Z 77,A -76.1324,B 24.9035,C -2.2683,E1 25.053,E2 520.416} C_DIS
LIN {X 20.3737,Y -65.0267,Z 77,A -78.5971,B 24.9042,C -2.26,E1 25.0464,E2 522.8955} C_DIS
LIN {X 18.1843,Y -65.6736,Z 77,A -80.7373,B 24.9048,C -2.2525,E1 25.0406,E2 525.0502} C_DIS
LIN {X 15.1309,Y -66.4426,Z 77,A -83.0606,B 24.9044,C -2.258,E1 25.0343,E2 527.357} C_DIS
LIN {X 12.6084,Y -66.9674,Z 77,A -85.3004,B 24.9047,C -2.2543,E1 25.0282,E2 529.6029} C_DIS
LIN {X 10.0091,Y -67.4055,Z 77,A -87.4991,B 24.9047,C -2.2532,E1 25.0221,E2 531.8022} C_DIS
LIN {X 7.5066,Y -67.7299,Z 77,A -89.6191,B 24.9049,C -2.2519,E1 25.0162,E2 533.9235} C_DIS
LIN {X 4.8684,Y -67.9698,Z 77,A -91.9748,B 24.9052,C -2.2477,E1 25.0097,E2 536.288} C_DIS
LIN {X 1.7763,Y -68.121,Z 77,A -94.4775,B 24.9051,C -2.2492,E1 25.0027,E2 538.7864} C_DIS
LIN {X 1.7763,Y -68.121,Z 77,A -94.4775,B 24.9051,C -2.2492,E1 25.0027,E2 538.7864} C_DIS
Enddeposition()
LIN {X 0.4221,Y -67.1891,Z 77,A -94.957,B 24.9023,C -2.2815,E1 25.0016,E2 539.1893} C_DIS
Startdeposition()
$VEL.CP = VEL_PRINT
LIN {X 2.4656,Y -67.1471,Z 77,A -92.6657,B 24.9012,C -2.2953,E1 25.0081,E2 536.8657} C_DIS
LIN {X 4.9301,Y -67.0113,Z 77,A -90.7689,B 24.9015,C -2.2911,E1 25.0133,E2 534.9796} C_DIS
LIN {X 7.4117,Y -66.7824,Z 77,A -88.4421,B 24.901,C -2.2973,E1 25.0198,E2 532.6398} C_DIS
LIN {X 9.8593,Y -66.4652,Z 77,A -86.3384,B 24.9009,C -2.2987,E1 25.0256,E2 530.5346} C_DIS
LIN {X 12.4304,Y -66.0319,Z 77,A -84.1679,B 24.9009,C -2.2991,E1 25.0316,E2 528.3654} C_DIS
LIN {X 15.3768,Y -65.4085,Z 77,A -81.751,B 24.9009,C -2.2977,E1 25.0382,E2 525.9551} C_DIS
LIN {X 17.9018,Y -64.7637,Z 77,A -79.335,B 24.9003,C -2.3048,E1 25.0447,E2 523.5259} C_DIS
LIN {X 20.2975,Y -64.0533,Z 77,A -77.4112,B 24.9006,C -2.3021,E1 25.0498,E2 521.6122} C_DIS
LIN {X 22.6479,Y -63.2605,Z 77,A -75.1089,B 24.8999,C -2.3095,E1 25.0559,E2 519.297} C_DIS
LIN {X 25.0826,Y -62.3345,Z 77,A -72.9422,B 24.8998,C -2.3112,E1 25.0616,E2 517.1311} C_DIS
LIN {X 27.8487,Y -61.1488,Z 77,A -70.615,B 24.9,C -2.3089,E1 25.0675,E2 514.815} C_DIS
LIN {X 30.0733,Y -60.0859,Z 77,A -68.4326,B 24.8995,C -2.3143,E1 25.073,E2 512.6255} C_DIS
LIN {X 32.3787,Y -58.8763,Z 77,A -66.2454,B 24.8993,C -2.3172,E1 25.0784,E2 510.4377} C_DIS
LIN {X 34.5573,Y -57.6247,Z 77,A -63.879,B 24.8984,C -2.3268,E1 25.0841,E2 508.0556} C_DIS
LIN {X 37.3142,Y -55.879,Z 77,A -61.1158,B 24.898,C -2.3317,E1 25.0906,E2 505.29} C_DIS
LIN {X 40.1383,Y -53.8855,Z 77,A -58.2365,B 24.8976,C -2.3359,E1 25.0971,E2 502.4109} C_DIS
LIN {X 42.5684,Y -51.9875,Z 77,A -55.6157,B 24.8971,C -2.3414,E1 25.1028,E2 499.787} C_DIS
LIN {X 44.8208,Y -50.0575,Z 77,A -53.0512,B 24.8966,C -2.348,E1 25.1082,E2 497.2168} C_DIS
LIN {X 46.9264,Y -48.0909,Z 77,A -50.5926,B 24.896,C -2.3538,E1 25.1132,E2 494.7547} C_DIS
LIN {X 48.9916,Y -45.9835,Z 77,A -48.1024,B 24.8955,C -2.3593,E1 25.118,E2 492.2623} C_DIS
LIN {X 51.0947,Y -43.6348,Z 77,A -45.5362,B 24.8952,C -2.3629,E1 25.1227,E2 489.6991} C_DIS
LIN {X 52.9719,Y -41.3376,Z 77,A -42.9178,B 24.8944,C -2.3719,E1 25.1273,E2 487.0718} C_DIS
LIN {X 54.4552,Y -39.3632,Z 77,A -40.8241,B 24.894,C -2.3772,E1 25.1307,E2 484.9756} C_DIS
LIN {X 55.9415,Y -37.2193,Z 77,A -38.6471,B 24.8935,C -2.3821,E1 25.1341,E2 482.7979} C_DIS
LIN {X 57.6188,Y -34.567,Z 77,A -35.9681,B 24.8928,C -2.3897,E1 25.1381,E2 480.1145} C_DIS
LIN {X 59.1119,Y -31.9445,Z 77,A -33.5565,B 24.8926,C -2.3928,E1 25.1413,E2 477.7082} C_DIS
LIN {X 60.3796,Y -29.4809,Z 77,A -31.3499,B 24.8923,C -2.3955,E1 25.1441,E2 475.5069} C_DIS
LIN {X 61.148,Y -27.8504,Z 77,A -29.575,B 24.8913,C -2.4065,E1 25.1462,E2 473.7156} C_DIS
LIN {X 62.3339,Y -25.084,Z 77,A -27.2559,B 24.8913,C -2.4075,E1 25.1487,E2 471.4068} C_DIS
LIN {X 63.2123,Y -22.78,Z 77,A -25.1663,B 24.8907,C -2.4136,E1 25.1507,E2 469.3146} C_DIS
LIN {X 63.9025,Y -20.7636,Z 77,A -23.1587,B 24.8897,C -2.4243,E1 25.1525,E2 467.2929} C_DIS
LIN {X 64.7582,Y -17.922,Z 77,A -20.5625,B 24.8888,C -2.4339,E1 25.1545,E2 464.6888} C_DIS
LIN {X 65.3767,Y -15.5146,Z 77,A -18.466,B 24.8883,C -2.44,E1 25.1559,E2 462.5902} C_DIS
LIN {X 65.9024,Y -13.1033,Z 77,A -16.5772,B 24.8882,C -2.4407,E1 25.157,E2 460.7105} C_DIS
LIN {X 66.3392,Y -10.6741,Z 77,A -14.2834,B 24.8871,C -2.4525,E1 25.1581,E2 458.4024} C_DIS
LIN {X 66.6864,Y -8.2304,Z 77,A -12.1928,B 24.8865,C -2.4588,E1 25.1588,E2 456.3093} C_DIS
LIN {X 66.9448,Y -5.7635,Z 77,A -10.0899,B 24.8859,C -2.4652,E1 25.1593,E2 454.2038} C_DIS
LIN {X 67.1118,Y -3.2896,Z 77,A -7.9954,B 24.8854,C -2.4714,E1 25.1597,E2 452.1071} C_DIS
LIN {X 67.1888,Y -0.5806,Z 77,A -5.7238,B 24.8848,C -2.4777,E1 25.1597,E2 449.8341} C_DIS
LIN {X 67.147,Y 2.4692,Z 77,A -3.1157,B 24.884,C -2.4861,E1 25.1596,E2 447.2217} C_DIS
LIN {X 66.9838,Y 5.2757,Z 77,A -0.7972,B 24.8835,C -2.4915,E1 25.1591,E2 444.9041} C_DIS
LIN {X 66.6869,Y 8.2272,Z 77,A 1.5725,B 24.8831,C -2.4951,E1 25.1584,E2 442.54} C_DIS
LIN {X 66.3397,Y 10.6711,Z 77,A 3.8674,B 24.882,C -2.5068,E1 25.1574,E2 440.231} C_DIS
LIN {X 65.9029,Y 13.1005,Z 77,A 5.9091,B 24.8816,C -2.5115,E1 25.1564,E2 438.19} C_DIS
LIN {X 65.3402,Y 15.6648,Z 77,A 8.1304,B 24.881,C -2.5179,E1 25.155,E2 435.9666} C_DIS
LIN {X 64.5721,Y 18.5788,Z 77,A 10.5454,B 24.8807,C -2.5214,E1 25.1532,E2 433.557} C_DIS
LIN {X 63.7966,Y 21.0905,Z 77,A 12.9865,B 24.8795,C -2.5334,E1 25.1511,E2 431.1015} C_DIS
LIN {X 62.7412,Y 24.0472,Z 77,A 15.3381,B 24.8796,C -2.5325,E1 25.1489,E2 428.7652} C_DIS
LIN {X 61.7657,Y 26.4538,Z 77,A 17.8503,B 24.8782,C -2.5467,E1 25.1461,E2 426.2331} C_DIS
LIN {X 60.405,Y 29.4283,Z 77,A 20.3939,B 24.8782,C -2.5479,E1 25.1431,E2 423.7004} C_DIS
LIN {X 59.259,Y 31.6732,Z 77,A 22.7299,B 24.8771,C -2.5587,E1 25.1401,E2 421.3512} C_DIS
LIN {X 58.0559,Y 33.828,Z 77,A 24.8443,B 24.8765,C -2.5645,E1 25.1371,E2 419.234} C_DIS
LIN {X 56.3963,Y 36.5265,Z 77,A 27.2241,B 24.8767,C -2.563,E1 25.1336,E2 416.8698} C_DIS
LIN {X 54.9431,Y 38.6791,Z 77,A 29.7399,B 24.8754,C -2.5764,E1 25.1296,E2 414.3346} C_DIS
LIN {X 53.2409,Y 40.9885,Z 77,A 32.1384,B 24.8749,C -2.5811,E1 25.1256,E2 411.9366} C_DIS
LIN {X 51.4582,Y 43.2068,Z 77,A 34.4876,B 24.8746,C -2.5847,E1 25.1214,E2 409.5898} C_DIS
LIN {X 49.5579,Y 45.3727,Z 77,A 36.89,B 24.8742,C -2.5887,E1 25.1169,E2 407.1884} C_DIS
LIN {X 47.5082,Y 47.5163,Z 77,A 39.5331,B 24.8734,C -2.597,E1 25.1118,E2 404.537} C_DIS
LIN {X 45.4355,Y 49.5002,Z 77,A 41.9535,B 24.873,C -2.6013,E1 25.1068,E2 402.1163} C_DIS
LIN {X 43.2333,Y 51.4362,Z 77,A 44.4676,B 24.8725,C -2.6064,E1 25.1015,E2 399.6} C_DIS
LIN {X 40.6877,Y 53.4728,Z 77,A 47.215,B 24.872,C -2.6106,E1 25.0954,E2 396.8529} C_DIS
LIN {X 38.6953,Y 54.9317,Z 77,A 49.3126,B 24.8717,C -2.6139,E1 25.0907,E2 394.7547} C_DIS
LIN {X 36.6347,Y 56.3269,Z 77,A 51.4233,B 24.8714,C -2.617,E1 25.0857,E2 392.6437} C_DIS
LIN {X 34.5481,Y 57.6303,Z 77,A 53.5171,B 24.8711,C -2.62,E1 25.0807,E2 390.5494} C_DIS
LIN {X 32.4157,Y 58.856,Z 77,A 55.6062,B 24.8709,C -2.6226,E1 25.0757,E2 388.4601} C_DIS
LIN {X 30.2093,Y 60.0185,Z 77,A 57.7299,B 24.8706,C -2.6252,E1 25.0704,E2 386.3361} C_DIS
LIN {X 27.8575,Y 61.1448,Z 77,A 59.8987,B 24.8705,C -2.6265,E1 25.0649,E2 384.1699} C_DIS
LIN {X 25.0893,Y 62.3318,Z 77,A 62.2276,B 24.8708,C -2.6232,E1 25.0589,E2 381.8541} C_DIS
LIN {X 22.8303,Y 63.1939,Z 77,A 64.3025,B 24.8706,C -2.6255,E1 25.0535,E2 379.7783} C_DIS
LIN {X 20.4443,Y 64.0059,Z 77,A 66.5235,B 24.8702,C -2.6289,E1 25.0476,E2 377.5534} C_DIS
LIN {X 17.9385,Y 64.7535,Z 77,A 68.8639,B 24.8698,C -2.6332,E1 25.0413,E2 375.2069} C_DIS
LIN {X 15.5263,Y 65.374,Z 77,A 71.0618,B 24.8695,C -2.6362,E1 25.0353,E2 373.0051} C_DIS
LIN {X 13.1135,Y 65.9004,Z 77,A 72.9571,B 24.8699,C -2.632,E1 25.0302,E2 371.1219} C_DIS
LIN {X 10.6832,Y 66.3377,Z 77,A 75.1444,B 24.8697,C -2.6347,E1 25.0241,E2 368.9306} C_DIS
LIN {X 8.2236,Y 66.6873,Z 77,A 77.3868,B 24.8693,C -2.6381,E1 25.0179,E2 366.6819} C_DIS
LIN {X 5.7679,Y 66.9444,Z 77,A 79.4923,B 24.8693,C -2.6383,E1 25.0121,E2 364.5771} C_DIS
LIN {X 3.3046,Y 67.1111,Z 77,A 81.34,B 24.8699,C -2.6322,E1 25.007,E2 362.7447} C_DIS
LIN {X 0.8372,Y 67.1872,Z 77,A 83.7068,B 24.8693,C -2.6381,E1 25.0003,E2 360.3642} C_DIS
LIN {X -1.6485,Y 67.1722,Z 77,A 85.8247,B 24.8693,C -2.6375,E1 24.9944,E2 358.2476} C_DIS
LIN {X -4.1157,Y 67.0663,Z 77,A 87.9318,B 24.8695,C -2.6368,E1 24.9885,E2 356.1417} C_DIS
LIN {X -6.7156,Y 66.8553,Z 77,A 90.1113,B 24.8697,C -2.6347,E1 24.9825,E2 353.966} C_DIS
LIN {X -9.1868,Y 66.5607,Z 77,A 92.2324,B 24.8697,C -2.6334,E1 24.9766,E2 351.8465} C_DIS
LIN {X -12.162,Y 66.0819,Z 77,A 94.6919,B 24.8702,C -2.629,E1 24.9699,E2 349.395} C_DIS
LIN {X -14.7464,Y 65.5542,Z 77,A 97.1049,B 24.87,C -2.6308,E1 24.9633,E2 346.9748} C_DIS
Enddeposition()
END
